KUKA KRL data list: CNC1.dat

&ACCESS RV
DEFDAT CNC1 Public
DECL GLOBAL FRAME gfCNCPoint1[30000]


gfCNCPoint1[1] = {X 300.0000, Y -7.9400, Z 3.0000, A 0.000, B 0.000, C 0.000 }
gfCNCPoint1[2] = {X 300.0000, Y -7.9400, Z 0.0000, A 0.000, B 0.000, C 0.000 }
gfCNCPoint1[3] = {X 300.0000, Y -1.5400, Z 0.0000, A 0.000, B 0.000, C 0.000 }
gfCNCPoint1[4] = {X 0.0000, Y -1.5400, Z 0.0000, A 0.000, B 0.000, C 0.000 }
gfCNCPoint1[5] = {X -1.5400, Y 0.0000, Z 0.0000, A 0.000, B 0.000, C 0.000 }
gfCNCPoint1[6] = {X -1.5400, Y 100.0000, Z 0.0000, A 0.000, B 0.000, C 0.000 }
gfCNCPoint1[7] = {X 0.0000, Y 101.5400, Z 0.0000, A 0.000, B 0.000, C 0.000 }
gfCNCPoint1[8] = {X 600.0000, Y 101.5400, Z 0.0000, A 0.000, B 0.000, C 0.000 }
gfCNCPoint1[9] = {X 601.5400, Y 100.0000, Z 0.0000, A 0.000, B 0.000, C 0.000 }
gfCNCPoint1[10] = {X 601.5400, Y 0.0000, Z 0.0000, A 0.000, B 0.000, C 0.000 }
gfCNCPoint1[11] = {X 600.0000, Y -1.5400, Z 0.0000, A 0.000, B 0.000, C 0.000 }
gfCNCPoint1[12] = {X 300.0000, Y -1.5400, Z 0.0000, A 0.000, B 0.000, C 0.000 }
gfCNCPoint1[13] = {X 300.0000, Y 0.8600, Z 0.0000, A 0.000, B 0.000, C 0.000 }
gfCNCPoint1[14] = {X 0.8600, Y 0.8600, Z 0.0000, A 0.000, B 0.000, C 0.000 }
gfCNCPoint1[15] = {X 0.8600, Y 99.1400, Z 0.0000, A 0.000, B 0.000, C 0.000 }
gfCNCPoint1[16] = {X 599.1400, Y 99.1400, Z 0.0000, A 0.000, B 0.000, C 0.000 }
gfCNCPoint1[17] = {X 599.1400, Y 0.8600, Z 0.0000, A 0.000, B 0.000, C 0.000 }
gfCNCPoint1[18] = {X 300.0000, Y 0.8600, Z 0.0000, A 0.000, B 0.000, C 0.000 }
gfCNCPoint1[19] = {X 300.0000, Y 3.2600, Z 0.0000, A 0.000, B 0.000, C 0.000 }
gfCNCPoint1[20] = {X 3.2600, Y 3.2600, Z 0.0000, A 0.000, B 0.000, C 0.000 }
gfCNCPoint1[21] = {X 3.2600, Y 96.7400, Z 0.0000, A 0.000, B 0.000, C 0.000 }
gfCNCPoint1[22] = {X 596.7400, Y 96.7400, Z 0.0000, A 0.000, B 0.000, C 0.000 }
gfCNCPoint1[23] = {X 596.7400, Y 3.2600, Z 0.0000, A 0.000, B 0.000, C 0.000 }
gfCNCPoint1[24] = {X 300.0000, Y 3.2600, Z 0.0000, A 0.000, B 0.000, C 0.000 }
gfCNCPoint1[25] = {X 300.0000, Y 5.6600, Z 0.0000, A 0.000, B 0.000, C 0.000 }
gfCNCPoint1[26] = {X 5.6600, Y 5.6600, Z 0.0000, A 0.000, B 0.000, C 0.000 }
gfCNCPoint1[27] = {X 5.6600, Y 94.3400, Z 0.0000, A 0.000, B 0.000, C 0.000 }
gfCNCPoint1[28] = {X 594.3400, Y 94.3400, Z 0.0000, A 0.000, B 0.000, C 0.000 }
gfCNCPoint1[29] = {X 594.3400, Y 5.6600, Z 0.0000, A 0.000, B 0.000, C 0.000 }
gfCNCPoint1[30] = {X 300.0000, Y 5.6600, Z 0.0000, A 0.000, B 0.000, C 0.000 }
gfCNCPoint1[31] = {X 300.0000, Y 8.0600, Z 0.0000, A 0.000, B 0.000, C 0.000 }
gfCNCPoint1[32] = {X 8.0600, Y 8.0600, Z 0.0000, A 0.000, B 0.000, C 0.000 }
gfCNCPoint1[33] = {X 8.0600, Y 91.9400, Z 0.0000, A 0.000, B 0.000, C 0.000 }
gfCNCPoint1[34] = {X 591.9400, Y 91.9400, Z 0.0000, A 0.000, B 0.000, C 0.000 }
gfCNCPoint1[35] = {X 591.9400, Y 8.0600, Z 0.0000, A 0.000, B 0.000, C 0.000 }
gfCNCPoint1[36] = {X 300.0000, Y 8.0600, Z 0.0000, A 0.000, B 0.000, C 0.000 }
gfCNCPoint1[37] = {X 300.0000, Y 10.4600, Z 0.0000, A 0.000, B 0.000, C 0.000 }
gfCNCPoint1[38] = {X 10.4600, Y 10.4600, Z 0.0000, A 0.000, B 0.000, C 0.000 }
gfCNCPoint1[39] = {X 10.4600, Y 89.5400, Z 0.0000, A 0.000, B 0.000, C 0.000 }
gfCNCPoint1[40] = {X 589.5400, Y 89.5400, Z 0.0000, A 0.000, B 0.000, C 0.000 }
gfCNCPoint1[41] = {X 589.5400, Y 10.4600, Z 0.0000, A 0.000, B 0.000, C 0.000 }
gfCNCPoint1[42] = {X 300.0000, Y 10.4600, Z 0.0000, A 0.000, B 0.000, C 0.000 }
gfCNCPoint1[43] = {X 300.0000, Y 12.8600, Z 0.0000, A 0.000, B 0.000, C 0.000 }
gfCNCPoint1[44] = {X 12.8600, Y 12.8600, Z 0.0000, A 0.000, B 0.000, C 0.000 }
gfCNCPoint1[45] = {X 12.8600, Y 87.1400, Z 0.0000, A 0.000, B 0.000, C 0.000 }
gfCNCPoint1[46] = {X 587.1400, Y 87.1400, Z 0.0000, A 0.000, B 0.000, C 0.000 }
gfCNCPoint1[47] = {X 587.1400, Y 12.8600, Z 0.0000, A 0.000, B 0.000, C 0.000 }
gfCNCPoint1[48] = {X 300.0000, Y 12.8600, Z 0.0000, A 0.000, B 0.000, C 0.000 }
gfCNCPoint1[49] = {X 300.0000, Y 15.2600, Z 0.0000, A 0.000, B 0.000, C 0.000 }
gfCNCPoint1[50] = {X 15.2600, Y 15.2600, Z 0.0000, A 0.000, B 0.000, C 0.000 }
gfCNCPoint1[51] = {X 15.2600, Y 84.7400, Z 0.0000, A 0.000, B 0.000, C 0.000 }
gfCNCPoint1[52] = {X 584.7400, Y 84.7400, Z 0.0000, A 0.000, B 0.000, C 0.000 }
gfCNCPoint1[53] = {X 584.7400, Y 15.2600, Z 0.0000, A 0.000, B 0.000, C 0.000 }
gfCNCPoint1[54] = {X 300.0000, Y 15.2600, Z 0.0000, A 0.000, B 0.000, C 0.000 }
gfCNCPoint1[55] = {X 300.0000, Y 17.6600, Z 0.0000, A 0.000, B 0.000, C 0.000 }
gfCNCPoint1[56] = {X 17.6600, Y 17.6600, Z 0.0000, A 0.000, B 0.000, C 0.000 }
gfCNCPoint1[57] = {X 17.6600, Y 82.3400, Z 0.0000, A 0.000, B 0.000, C 0.000 }
gfCNCPoint1[58] = {X 582.3400, Y 82.3400, Z 0.0000, A 0.000, B 0.000, C 0.000 }
gfCNCPoint1[59] = {X 582.3400, Y 17.6600, Z 0.0000, A 0.000, B 0.000, C 0.000 }
gfCNCPoint1[60] = {X 300.0000, Y 17.6600, Z 0.0000, A 0.000, B 0.000, C 0.000 }
gfCNCPoint1[61] = {X 300.0000, Y 20.0600, Z 0.0000, A 0.000, B 0.000, C 0.000 }
gfCNCPoint1[62] = {X 20.0600, Y 20.0600, Z 0.0000, A 0.000, B 0.000, C 0.000 }
gfCNCPoint1[63] = {X 20.0600, Y 79.9400, Z 0.0000, A 0.000, B 0.000, C 0.000 }
gfCNCPoint1[64] = {X 579.9400, Y 79.9400, Z 0.0000, A 0.000, B 0.000, C 0.000 }
gfCNCPoint1[65] = {X 579.9400, Y 20.0600, Z 0.0000, A 0.000, B 0.000, C 0.000 }
gfCNCPoint1[66] = {X 300.0000, Y 20.0600, Z 0.0000, A 0.000, B 0.000, C 0.000 }
gfCNCPoint1[67] = {X 300.0000, Y 22.4600, Z 0.0000, A 0.000, B 0.000, C 0.000 }
gfCNCPoint1[68] = {X 22.4600, Y 22.4600, Z 0.0000, A 0.000, B 0.000, C 0.000 }
gfCNCPoint1[69] = {X 22.4600, Y 77.5400, Z 0.0000, A 0.000, B 0.000, C 0.000 }
gfCNCPoint1[70] = {X 577.5400, Y 77.5400, Z 0.0000, A 0.000, B 0.000, C 0.000 }
gfCNCPoint1[71] = {X 577.5400, Y 22.4600, Z 0.0000, A 0.000, B 0.000, C 0.000 }
gfCNCPoint1[72] = {X 300.0000, Y 22.4600, Z 0.0000, A 0.000, B 0.000, C 0.000 }
gfCNCPoint1[73] = {X 300.0000, Y 24.8600, Z 0.0000, A 0.000, B 0.000, C 0.000 }
gfCNCPoint1[74] = {X 24.8600, Y 24.8600, Z 0.0000, A 0.000, B 0.000, C 0.000 }
gfCNCPoint1[75] = {X 24.8600, Y 75.1400, Z 0.0000, A 0.000, B 0.000, C 0.000 }
gfCNCPoint1[76] = {X 575.1400, Y 75.1400, Z 0.0000, A 0.000, B 0.000, C 0.000 }
gfCNCPoint1[77] = {X 575.1400, Y 24.8600, Z 0.0000, A 0.000, B 0.000, C 0.000 }
gfCNCPoint1[78] = {X 300.0000, Y 24.8600, Z 0.0000, A 0.000, B 0.000, C 0.000 }
gfCNCPoint1[79] = {X 300.0000, Y 27.2600, Z 0.0000, A 0.000, B 0.000, C 0.000 }
gfCNCPoint1[80] = {X 27.2600, Y 27.2600, Z 0.0000, A 0.000, B 0.000, C 0.000 }
gfCNCPoint1[81] = {X 27.2600, Y 72.7400, Z 0.0000, A 0.000, B 0.000, C 0.000 }
gfCNCPoint1[82] = {X 572.7400, Y 72.7400, Z 0.0000, A 0.000, B 0.000, C 0.000 }
gfCNCPoint1[83] = {X 572.7400, Y 27.2600, Z 0.0000, A 0.000, B 0.000, C 0.000 }
gfCNCPoint1[84] = {X 300.0000, Y 27.2600, Z 0.0000, A 0.000, B 0.000, C 0.000 }
gfCNCPoint1[85] = {X 300.0000, Y 29.6600, Z 0.0000, A 0.000, B 0.000, C 0.000 }
gfCNCPoint1[86] = {X 29.6600, Y 29.6600, Z 0.0000, A 0.000, B 0.000, C 0.000 }
gfCNCPoint1[87] = {X 29.6600, Y 70.3400, Z 0.0000, A 0.000, B 0.000, C 0.000 }
gfCNCPoint1[88] = {X 570.3400, Y 70.3400, Z 0.0000, A 0.000, B 0.000, C 0.000 }
gfCNCPoint1[89] = {X 570.3400, Y 29.6600, Z 0.0000, A 0.000, B 0.000, C 0.000 }
gfCNCPoint1[90] = {X 300.0000, Y 29.6600, Z 0.0000, A 0.000, B 0.000, C 0.000 }
gfCNCPoint1[91] = {X 300.0000, Y 32.0600, Z 0.0000, A 0.000, B 0.000, C 0.000 }
gfCNCPoint1[92] = {X 32.0600, Y 32.0600, Z 0.0000, A 0.000, B 0.000, C 0.000 }
gfCNCPoint1[93] = {X 32.0600, Y 67.9400, Z 0.0000, A 0.000, B 0.000, C 0.000 }
gfCNCPoint1[94] = {X 567.9400, Y 67.9400, Z 0.0000, A 0.000, B 0.000, C 0.000 }
gfCNCPoint1[95] = {X 567.9400, Y 32.0600, Z 0.0000, A 0.000, B 0.000, C 0.000 }
gfCNCPoint1[96] = {X 300.0000, Y 32.0600, Z 0.0000, A 0.000, B 0.000, C 0.000 }
gfCNCPoint1[97] = {X 300.0000, Y 34.4600, Z 0.0000, A 0.000, B 0.000, C 0.000 }
gfCNCPoint1[98] = {X 34.4600, Y 34.4600, Z 0.0000, A 0.000, B 0.000, C 0.000 }
gfCNCPoint1[99] = {X 34.4600, Y 65.5400, Z 0.0000, A 0.000, B 0.000, C 0.000 }
gfCNCPoint1[100] = {X 565.5400, Y 65.5400, Z 0.0000, A 0.000, B 0.000, C 0.000 }
gfCNCPoint1[101] = {X 565.5400, Y 34.4600, Z 0.0000, A 0.000, B 0.000, C 0.000 }
gfCNCPoint1[102] = {X 300.0000, Y 34.4600, Z 0.0000, A 0.000, B 0.000, C 0.000 }
gfCNCPoint1[103] = {X 300.0000, Y 36.8600, Z 0.0000, A 0.000, B 0.000, C 0.000 }
gfCNCPoint1[104] = {X 36.8600, Y 36.8600, Z 0.0000, A 0.000, B 0.000, C 0.000 }
gfCNCPoint1[105] = {X 36.8600, Y 63.1400, Z 0.0000, A 0.000, B 0.000, C 0.000 }
gfCNCPoint1[106] = {X 563.1400, Y 63.1400, Z 0.0000, A 0.000, B 0.000, C 0.000 }
gfCNCPoint1[107] = {X 563.1400, Y 36.8600, Z 0.0000, A 0.000, B 0.000, C 0.000 }
gfCNCPoint1[108] = {X 300.0000, Y 36.8600, Z 0.0000, A 0.000, B 0.000, C 0.000 }
gfCNCPoint1[109] = {X 300.0000, Y 39.2600, Z 0.0000, A 0.000, B 0.000, C 0.000 }
gfCNCPoint1[110] = {X 39.2600, Y 39.2600, Z 0.0000, A 0.000, B 0.000, C 0.000 }
gfCNCPoint1[111] = {X 39.2600, Y 60.7400, Z 0.0000, A 0.000, B 0.000, C 0.000 }
gfCNCPoint1[112] = {X 560.7400, Y 60.7400, Z 0.0000, A 0.000, B 0.000, C 0.000 }
gfCNCPoint1[113] = {X 560.7400, Y 39.2600, Z 0.0000, A 0.000, B 0.000, C 0.000 }
gfCNCPoint1[114] = {X 300.0000, Y 39.2600, Z 0.0000, A 0.000, B 0.000, C 0.000 }
gfCNCPoint1[115] = {X 300.0000, Y 41.6600, Z 0.0000, A 0.000, B 0.000, C 0.000 }
gfCNCPoint1[116] = {X 41.6600, Y 41.6600, Z 0.0000, A 0.000, B 0.000, C 0.000 }
gfCNCPoint1[117] = {X 41.6600, Y 58.3400, Z 0.0000, A 0.000, B 0.000, C 0.000 }
gfCNCPoint1[118] = {X 558.3400, Y 58.3400, Z 0.0000, A 0.000, B 0.000, C 0.000 }
gfCNCPoint1[119] = {X 558.3400, Y 41.6600, Z 0.0000, A 0.000, B 0.000, C 0.000 }
gfCNCPoint1[120] = {X 300.0000, Y 41.6600, Z 0.0000, A 0.000, B 0.000, C 0.000 }
gfCNCPoint1[121] = {X 300.0000, Y 44.0600, Z 0.0000, A 0.000, B 0.000, C 0.000 }
gfCNCPoint1[122] = {X 44.0600, Y 44.0600, Z 0.0000, A 0.000, B 0.000, C 0.000 }
gfCNCPoint1[123] = {X 44.0600, Y 55.9400, Z 0.0000, A 0.000, B 0.000, C 0.000 }
gfCNCPoint1[124] = {X 555.9400, Y 55.9400, Z 0.0000, A 0.000, B 0.000, C 0.000 }
gfCNCPoint1[125] = {X 555.9400, Y 44.0600, Z 0.0000, A 0.000, B 0.000, C 0.000 }
gfCNCPoint1[126] = {X 300.0000, Y 44.0600, Z 0.0000, A 0.000, B 0.000, C 0.000 }
gfCNCPoint1[127] = {X 300.0000, Y 46.4600, Z 0.0000, A 0.000, B 0.000, C 0.000 }
gfCNCPoint1[128] = {X 46.4600, Y 46.4600, Z 0.0000, A 0.000, B 0.000, C 0.000 }
gfCNCPoint1[129] = {X 46.4600, Y 53.5400, Z 0.0000, A 0.000, B 0.000, C 0.000 }
gfCNCPoint1[130] = {X 553.5400, Y 53.5400, Z 0.0000, A 0.000, B 0.000, C 0.000 }
gfCNCPoint1[131] = {X 553.5400, Y 46.4600, Z 0.0000, A 0.000, B 0.000, C 0.000 }
gfCNCPoint1[132] = {X 300.0000, Y 46.4600, Z 0.0000, A 0.000, B 0.000, C 0.000 }
gfCNCPoint1[133] = {X 300.0000, Y 48.8600, Z 0.0000, A 0.000, B 0.000, C 0.000 }
gfCNCPoint1[134] = {X 48.8600, Y 48.8600, Z 0.0000, A 0.000, B 0.000, C 0.000 }
gfCNCPoint1[135] = {X 48.8600, Y 51.1400, Z 0.0000, A 0.000, B 0.000, C 0.000 }
gfCNCPoint1[136] = {X 551.1400, Y 51.1400, Z 0.0000, A 0.000, B 0.000, C 0.000 }
gfCNCPoint1[137] = {X 551.1400, Y 48.8600, Z 0.0000, A 0.000, B 0.000, C 0.000 }
gfCNCPoint1[138] = {X 300.0000, Y 48.8600, Z 0.0000, A 0.000, B 0.000, C 0.000 }
gfCNCPoint1[139] = {X 300.0000, Y 44.8600, Z 0.0000, A 0.000, B 0.000, C 0.000 }
gfCNCPoint1[140] = {X 300.0000, Y 44.8600, Z 3.0000, A 0.000, B 0.000, C 0.000 }
gfCNCPoint1[141] = {X 300.0000, Y 44.8600, Z 10.0000, A 0.000, B 0.000, C 0.000 }
gfCNCPoint1[142] = {X 607.6965, Y 2.1256, Z 1.6667, A 0.000, B 0.000, C 0.000 }
gfCNCPoint1[143] = {X 607.6965, Y 2.1256, Z -1.3333, A 0.000, B 0.000, C 0.000 }
gfCNCPoint1[144] = {X 603.6965, Y 8.3207, Z -1.3333, A 0.000, B 0.000, C 0.000 }
gfCNCPoint1[145] = {X 603.3199, Y 8.8216, Z -1.3333, A 0.000, B 0.000, C 0.000 }
gfCNCPoint1[146] = {X 602.8760, Y 9.2640, Z -1.3333, A 0.000, B 0.000, C 0.000 }
gfCNCPoint1[147] = {X 602.8760, Y 40.7360, Z -1.3333, A 0.000, B 0.000, C 0.000 }
gfCNCPoint1[148] = {X 603.3199, Y 41.1783, Z -1.3333, A 0.000, B 0.000, C 0.000 }
gfCNCPoint1[149] = {X 603.6965, Y 41.6793, Z -1.3333, A 0.000, B 0.000, C 0.000 }
gfCNCPoint1[150] = {X 607.6965, Y 47.8744, Z -1.3333, A 0.000, B 0.000, C 0.000 }
gfCNCPoint1[151] = {X 607.6965, Y 47.8744, Z 1.6667, A 0.000, B 0.000, C 0.000 }
gfCNCPoint1[152] = {X 607.6965, Y 47.8744, Z 11.0000, A 0.000, B 0.000, C 0.000 }
gfCNCPoint1[153] = {X 607.6965, Y 1.5529, Z 11.0000, A 0.000, B 0.000, C 0.000 }
gfCNCPoint1[154] = {X 607.6965, Y 1.5529, Z 1.6667, A 0.000, B 0.000, C 0.000 }
gfCNCPoint1[155] = {X 607.6965, Y 1.5529, Z -1.3333, A 0.000, B 0.000, C 0.000 }
gfCNCPoint1[156] = {X 603.6965, Y 8.1703, Z -1.3333, A 0.000, B 0.000, C 0.000 }
gfCNCPoint1[157] = {X 603.2890, Y 8.7356, Z -1.3333, A 0.000, B 0.000, C 0.000 }
gfCNCPoint1[158] = {X 602.7960, Y 9.2281, Z -1.3333, A 0.000, B 0.000, C 0.000 }
gfCNCPoint1[159] = {X 602.7960, Y 40.7730, Z -1.3333, A 0.000, B 0.000, C 0.000 }
gfCNCPoint1[160] = {X 603.2890, Y 41.2652, Z -1.3333, A 0.000, B 0.000, C 0.000 }
gfCNCPoint1[161] = {X 603.6965, Y 41.8302, Z -1.3333, A 0.000, B 0.000, C 0.000 }
gfCNCPoint1[162] = {X 607.6965, Y 48.4430, Z -1.3333, A 0.000, B 0.000, C 0.000 }
gfCNCPoint1[163] = {X 607.6965, Y 48.4430, Z 1.6667, A 0.000, B 0.000, C 0.000 }
gfCNCPoint1[164] = {X 607.6965, Y 48.4430, Z 11.0000, A 0.000, B 0.000, C 0.000 }
gfCNCPoint1[165] = {X 607.6965, Y 0.8876, Z 11.0000, A 0.000, B 0.000, C 0.000 }
gfCNCPoint1[166] = {X 607.6965, Y 0.8876, Z 1.6667, A 0.000, B 0.000, C 0.000 }
gfCNCPoint1[167] = {X 607.6965, Y 0.8876, Z -1.3333, A 0.000, B 0.000, C 0.000 }
gfCNCPoint1[168] = {X 603.6965, Y 8.0114, Z -1.3333, A 0.000, B 0.000, C 0.000 }
gfCNCPoint1[169] = {X 603.2600, Y 8.6459, Z -1.3333, A 0.000, B 0.000, C 0.000 }
gfCNCPoint1[170] = {X 602.7160, Y 9.1909, Z -1.3333, A 0.000, B 0.000, C 0.000 }
gfCNCPoint1[171] = {X 602.7160, Y 40.8102, Z -1.3333, A 0.000, B 0.000, C 0.000 }
gfCNCPoint1[172] = {X 603.2600, Y 41.3549, Z -1.3333, A 0.000, B 0.000, C 0.000 }
gfCNCPoint1[173] = {X 603.6965, Y 41.9890, Z -1.3333, A 0.000, B 0.000, C 0.000 }
gfCNCPoint1[174] = {X 607.6965, Y 49.1072, Z -1.3333, A 0.000, B 0.000, C 0.000 }
gfCNCPoint1[175] = {X 607.6965, Y 49.1072, Z 1.6667, A 0.000, B 0.000, C 0.000 }
gfCNCPoint1[176] = {X 607.6965, Y 49.1072, Z 11.0000, A 0.000, B 0.000, C 0.000 }
gfCNCPoint1[177] = {X 607.6950, Y 0.0916, Z 11.0000, A 0.000, B 0.000, C 0.000 }
gfCNCPoint1[178] = {X 607.6950, Y 0.0916, Z 1.6667, A 0.000, B 0.000, C 0.000 }
gfCNCPoint1[179] = {X 607.6950, Y 0.0916, Z -1.3333, A 0.000, B 0.000, C 0.000 }
gfCNCPoint1[180] = {X 603.6965, Y 7.8427, Z -1.3333, A 0.000, B 0.000, C 0.000 }
gfCNCPoint1[181] = {X 603.2333, Y 8.5523, Z -1.3333, A 0.000, B 0.000, C 0.000 }
gfCNCPoint1[182] = {X 602.6360, Y 9.1532, Z -1.3333, A 0.000, B 0.000, C 0.000 }
gfCNCPoint1[183] = {X 602.6360, Y 40.8479, Z -1.3333, A 0.000, B 0.000, C 0.000 }
gfCNCPoint1[184] = {X 603.2333, Y 41.4485, Z -1.3333, A 0.000, B 0.000, C 0.000 }
gfCNCPoint1[185] = {X 603.6965, Y 42.1576, Z -1.3333, A 0.000, B 0.000, C 0.000 }
gfCNCPoint1[186] = {X 607.6965, Y 49.9047, Z -1.3333, A 0.000, B 0.000, C 0.000 }
gfCNCPoint1[187] = {X 607.6965, Y 49.9047, Z 1.6667, A 0.000, B 0.000, C 0.000 }
gfCNCPoint1[188] = {X 607.6965, Y 49.9047, Z 11.0000, A 0.000, B 0.000, C 0.000 }
gfCNCPoint1[189] = {X 607.6538, Y -0.8091, Z 11.0000, A 0.000, B 0.000, C 0.000 }
gfCNCPoint1[190] = {X 607.6538, Y -0.8091, Z 1.6667, A 0.000, B 0.000, C 0.000 }
gfCNCPoint1[191] = {X 607.6538, Y -0.8091, Z -1.3333, A 0.000, B 0.000, C 0.000 }
gfCNCPoint1[192] = {X 603.6965, Y 7.6611, Z -1.3333, A 0.000, B 0.000, C 0.000 }
gfCNCPoint1[193] = {X 603.2067, Y 8.4567, Z -1.3333, A 0.000, B 0.000, C 0.000 }
gfCNCPoint1[194] = {X 602.5488, Y 9.1200, Z -1.3333, A 0.000, B 0.000, C 0.000 }
gfCNCPoint1[195] = {X 602.5560, Y 9.1532, Z -1.3333, A 0.000, B 0.000, C 0.000 }
gfCNCPoint1[196] = {X 602.5560, Y 40.8856, Z -1.3333, A 0.000, B 0.000, C 0.000 }
gfCNCPoint1[197] = {X 602.6236, Y 40.9413, Z -1.3333, A 0.000, B 0.000, C 0.000 }
gfCNCPoint1[198] = {X 603.2364, Y 41.5815, Z -1.3333, A 0.000, B 0.000, C 0.000 }
gfCNCPoint1[199] = {X 603.6965, Y 42.3389, Z -1.3333, A 0.000, B 0.000, C 0.000 }
gfCNCPoint1[200] = {X 607.6965, Y 50.9003, Z -1.3333, A 0.000, B 0.000, C 0.000 }
gfCNCPoint1[201] = {X 607.6965, Y 50.9003, Z 1.6667, A 0.000, B 0.000, C 0.000 }
gfCNCPoint1[202] = {X 607.6965, Y 50.9003, Z 11.0000, A 0.000, B 0.000, C 0.000 }
gfCNCPoint1[203] = {X 607.4989, Y -1.7333, Z 11.0000, A 0.000, B 0.000, C 0.000 }
gfCNCPoint1[204] = {X 607.4989, Y -1.7333, Z 1.6667, A 0.000, B 0.000, C 0.000 }
gfCNCPoint1[205] = {X 607.4989, Y -1.7333, Z -1.3333, A 0.000, B 0.000, C 0.000 }
gfCNCPoint1[206] = {X 603.6965, Y 7.4625, Z -1.3333, A 0.000, B 0.000, C 0.000 }
gfCNCPoint1[207] = {X 603.3768, Y 8.0782, Z -1.3333, A 0.000, B 0.000, C 0.000 }
gfCNCPoint1[208] = {X 602.9556, Y 8.6294, Z -1.3333, A 0.000, B 0.000, C 0.000 }
gfCNCPoint1[209] = {X 602.4454, Y 9.0995, Z -1.3333, A 0.000, B 0.000, C 0.000 }
gfCNCPoint1[210] = {X 602.4760, Y 9.1532, Z -1.3333, A 0.000, B 0.000, C 0.000 }
gfCNCPoint1[211] = {X 602.4760, Y 40.9232, Z -1.3333, A 0.000, B 0.000, C 0.000 }
gfCNCPoint1[212] = {X 602.5724, Y 41.0028, Z -1.3333, A 0.000, B 0.000, C 0.000 }
gfCNCPoint1[213] = {X 603.2270, Y 41.7024, Z -1.3333, A 0.000, B 0.000, C 0.000 }
gfCNCPoint1[214] = {X 603.6965, Y 42.5375, Z -1.3333, A 0.000, B 0.000, C 0.000 }
gfCNCPoint1[215] = {X 607.6965, Y 52.2111, Z -1.3333, A 0.000, B 0.000, C 0.000 }
gfCNCPoint1[216] = {X 607.6965, Y 52.2111, Z 1.6667, A 0.000, B 0.000, C 0.000 }
gfCNCPoint1[217] = {X 607.6965, Y 52.2111, Z 11.0000, A 0.000, B 0.000, C 0.000 }
gfCNCPoint1[218] = {X 492.1926, Y 19.7807, Z 11.0000, A 0.000, B 0.000, C 0.000 }
gfCNCPoint1[219] = {X 492.1926, Y 19.7807, Z 2.5000, A 0.000, B 0.000, C 0.000 }
gfCNCPoint1[220] = {X 487.6645, Y 19.7797, Z 1.2867, A 0.000, B 0.000, C 0.000 }
gfCNCPoint1[221] = {X 486.9699, Y 19.7845, Z 1.1006, A 0.000, B 0.000, C 0.000 }
gfCNCPoint1[222] = {X 486.2675, Y 19.7831, Z 0.9124, A 0.000, B 0.000, C 0.000 }
gfCNCPoint1[223] = {X 485.4752, Y 19.8882, Z 0.6982, A 0.000, B 0.000, C 0.000 }
gfCNCPoint1[224] = {X 484.7975, Y 20.0727, Z 0.5100, A 0.000, B 0.000, C 0.000 }
gfCNCPoint1[225] = {X 484.6636, Y 20.1091, Z 0.4728, A 0.000, B 0.000, C 0.000 }
gfCNCPoint1[226] = {X 484.6335, Y 20.1374, Z 0.4618, A 0.000, B 0.000, C 0.000 }
gfCNCPoint1[227] = {X 484.5885, Y 20.2686, Z 0.4246, A 0.000, B 0.000, C 0.000 }
gfCNCPoint1[228] = {X 484.4391, Y 20.7049, Z 0.3010, A 0.000, B 0.000, C 0.000 }
gfCNCPoint1[229] = {X 484.4030, Y 21.9111, Z -0.0223, A 0.000, B 0.000, C 0.000 }
gfCNCPoint1[230] = {X 484.5262, Y 22.3556, Z -0.1459, A 0.000, B 0.000, C 0.000 }
gfCNCPoint1[231] = {X 484.6980, Y 22.4116, Z -0.1943, A 0.000, B 0.000, C 0.000 }
gfCNCPoint1[232] = {X 484.8776, Y 22.4314, Z -0.2427, A 0.000, B 0.000, C 0.000 }
gfCNCPoint1[233] = {X 486.0306, Y 22.5560, Z -0.5535, A 0.000, B 0.000, C 0.000 }
gfCNCPoint1[234] = {X 487.1449, Y 22.5560, Z -0.8521, A 0.000, B 0.000, C 0.000 }
gfCNCPoint1[235] = {X 488.9410, Y 22.5560, Z -1.3333, A 0.000, B 0.000, C 0.000 }
gfCNCPoint1[236] = {X 493.3690, Y 22.5560, Z -1.3333, A 0.000, B 0.000, C 0.000 }
gfCNCPoint1[237] = {X 493.3690, Y 19.7809, Z -1.3333, A 0.000, B 0.000, C 0.000 }
gfCNCPoint1[238] = {X 487.6645, Y 19.7797, Z -1.3333, A 0.000, B 0.000, C 0.000 }
gfCNCPoint1[239] = {X 486.9699, Y 19.7845, Z -1.3333, A 0.000, B 0.000, C 0.000 }
gfCNCPoint1[240] = {X 485.8740, Y 19.8557, Z -1.3333, A 0.000, B 0.000, C 0.000 }
gfCNCPoint1[241] = {X 484.7975, Y 20.0727, Z -1.3333, A 0.000, B 0.000, C 0.000 }
gfCNCPoint1[242] = {X 484.6687, Y 20.1447, Z -1.3333, A 0.000, B 0.000, C 0.000 }
gfCNCPoint1[243] = {X 484.5885, Y 20.2686, Z -1.3333, A 0.000, B 0.000, C 0.000 }
gfCNCPoint1[244] = {X 484.4277, Y 20.9554, Z -1.3333, A 0.000, B 0.000, C 0.000 }
gfCNCPoint1[245] = {X 484.4067, Y 21.6604, Z -1.3333, A 0.000, B 0.000, C 0.000 }
gfCNCPoint1[246] = {X 484.5262, Y 22.3556, Z -1.3333, A 0.000, B 0.000, C 0.000 }
gfCNCPoint1[247] = {X 484.7000, Y 22.4025, Z -1.3333, A 0.000, B 0.000, C 0.000 }
gfCNCPoint1[248] = {X 484.8776, Y 22.4314, Z -1.3333, A 0.000, B 0.000, C 0.000 }
gfCNCPoint1[249] = {X 486.0096, Y 22.5249, Z -1.3333, A 0.000, B 0.000, C 0.000 }
gfCNCPoint1[250] = {X 487.1449, Y 22.5560, Z -1.3333, A 0.000, B 0.000, C 0.000 }
gfCNCPoint1[251] = {X 488.9410, Y 22.5560, Z -1.3333, A 0.000, B 0.000, C 0.000 }
gfCNCPoint1[252] = {X 484.9562, Y 22.2874, Z -1.3333, A 0.000, B 0.000, C 0.000 }
gfCNCPoint1[253] = {X 488.9410, Y 22.6360, Z -1.3333, A 0.000, B 0.000, C 0.000 }
gfCNCPoint1[254] = {X 493.4490, Y 22.6360, Z -1.3333, A 0.000, B 0.000, C 0.000 }
gfCNCPoint1[255] = {X 493.4490, Y 19.7009, Z -1.3333, A 0.000, B 0.000, C 0.000 }
gfCNCPoint1[256] = {X 487.6642, Y 19.6997, Z -1.3333, A 0.000, B 0.000, C 0.000 }
gfCNCPoint1[257] = {X 486.9714, Y 19.7045, Z -1.3333, A 0.000, B 0.000, C 0.000 }
gfCNCPoint1[258] = {X 485.8642, Y 19.7763, Z -1.3333, A 0.000, B 0.000, C 0.000 }
gfCNCPoint1[259] = {X 484.7765, Y 19.9955, Z -1.3333, A 0.000, B 0.000, C 0.000 }
gfCNCPoint1[260] = {X 484.6139, Y 20.0863, Z -1.3333, A 0.000, B 0.000, C 0.000 }
gfCNCPoint1[261] = {X 484.5129, Y 20.2427, Z -1.3333, A 0.000, B 0.000, C 0.000 }
gfCNCPoint1[262] = {X 484.3466, Y 20.9591, Z -1.3333, A 0.000, B 0.000, C 0.000 }
gfCNCPoint1[263] = {X 484.3290, Y 21.6943, Z -1.3333, A 0.000, B 0.000, C 0.000 }
gfCNCPoint1[264] = {X 484.4607, Y 22.4179, Z -1.3333, A 0.000, B 0.000, C 0.000 }
gfCNCPoint1[265] = {X 484.6621, Y 22.4761, Z -1.3333, A 0.000, B 0.000, C 0.000 }
gfCNCPoint1[266] = {X 484.8689, Y 22.5109, Z -1.3333, A 0.000, B 0.000, C 0.000 }
gfCNCPoint1[267] = {X 486.0052, Y 22.6047, Z -1.3333, A 0.000, B 0.000, C 0.000 }
gfCNCPoint1[268] = {X 487.1449, Y 22.6360, Z -1.3333, A 0.000, B 0.000, C 0.000 }
gfCNCPoint1[269] = {X 488.9410, Y 22.6360, Z -1.3333, A 0.000, B 0.000, C 0.000 }
gfCNCPoint1[270] = {X 492.9257, Y 22.2874, Z -1.3333, A 0.000, B 0.000, C 0.000 }
gfCNCPoint1[271] = {X 484.9562, Y 22.3674, Z -1.3333, A 0.000, B 0.000, C 0.000 }
gfCNCPoint1[272] = {X 488.9410, Y 22.7160, Z -1.3333, A 0.000, B 0.000, C 0.000 }
gfCNCPoint1[273] = {X 493.5290, Y 22.7160, Z -1.3333, A 0.000, B 0.000, C 0.000 }
gfCNCPoint1[274] = {X 493.5290, Y 19.6209, Z -1.3333, A 0.000, B 0.000, C 0.000 }
gfCNCPoint1[275] = {X 487.6640, Y 19.6197, Z -1.3333, A 0.000, B 0.000, C 0.000 }
gfCNCPoint1[276] = {X 486.9712, Y 19.6245, Z -1.3333, A 0.000, B 0.000, C 0.000 }
gfCNCPoint1[277] = {X 485.8535, Y 19.6971, Z -1.3333, A 0.000, B 0.000, C 0.000 }
gfCNCPoint1[278] = {X 484.7555, Y 19.9183, Z -1.3333, A 0.000, B 0.000, C 0.000 }
gfCNCPoint1[279] = {X 484.5592, Y 20.0279, Z -1.3333, A 0.000, B 0.000, C 0.000 }
gfCNCPoint1[280] = {X 484.4372, Y 20.2167, Z -1.3333, A 0.000, B 0.000, C 0.000 }
gfCNCPoint1[281] = {X 484.2655, Y 20.9625, Z -1.3333, A 0.000, B 0.000, C 0.000 }
gfCNCPoint1[282] = {X 484.2514, Y 21.7276, Z -1.3333, A 0.000, B 0.000, C 0.000 }
gfCNCPoint1[283] = {X 484.3954, Y 22.4792, Z -1.3333, A 0.000, B 0.000, C 0.000 }
gfCNCPoint1[284] = {X 484.6243, Y 22.5494, Z -1.3333, A 0.000, B 0.000, C 0.000 }
gfCNCPoint1[285] = {X 484.8601, Y 22.5904, Z -1.3333, A 0.000, B 0.000, C 0.000 }
gfCNCPoint1[286] = {X 486.0008, Y 22.6846, Z -1.3333, A 0.000, B 0.000, C 0.000 }
gfCNCPoint1[287] = {X 487.1449, Y 22.7160, Z -1.3333, A 0.000, B 0.000, C 0.000 }
gfCNCPoint1[288] = {X 488.9410, Y 22.7160, Z -1.3333, A 0.000, B 0.000, C 0.000 }
gfCNCPoint1[289] = {X 492.9257, Y 22.3674, Z -1.3333, A 0.000, B 0.000, C 0.000 }
gfCNCPoint1[290] = {X 484.9562, Y 22.4474, Z -1.3333, A 0.000, B 0.000, C 0.000 }
gfCNCPoint1[291] = {X 488.9410, Y 22.7960, Z -1.3333, A 0.000, B 0.000, C 0.000 }
gfCNCPoint1[292] = {X 493.6090, Y 22.7960, Z -1.3333, A 0.000, B 0.000, C 0.000 }
gfCNCPoint1[293] = {X 493.6090, Y 19.5409, Z -1.3333, A 0.000, B 0.000, C 0.000 }
gfCNCPoint1[294] = {X 487.6637, Y 19.5397, Z -1.3333, A 0.000, B 0.000, C 0.000 }
gfCNCPoint1[295] = {X 486.9711, Y 19.5445, Z -1.3333, A 0.000, B 0.000, C 0.000 }
gfCNCPoint1[296] = {X 485.8428, Y 19.6178, Z -1.3333, A 0.000, B 0.000, C 0.000 }
gfCNCPoint1[297] = {X 484.7345, Y 19.8411, Z -1.3333, A 0.000, B 0.000, C 0.000 }
gfCNCPoint1[298] = {X 484.5045, Y 19.9696, Z -1.3333, A 0.000, B 0.000, C 0.000 }
gfCNCPoint1[299] = {X 484.3615, Y 20.1908, Z -1.3333, A 0.000, B 0.000, C 0.000 }
gfCNCPoint1[300] = {X 484.1846, Y 20.9657, Z -1.3333, A 0.000, B 0.000, C 0.000 }
gfCNCPoint1[301] = {X 484.1740, Y 21.7605, Z -1.3333, A 0.000, B 0.000, C 0.000 }
gfCNCPoint1[302] = {X 484.3303, Y 22.5398, Z -1.3333, A 0.000, B 0.000, C 0.000 }
gfCNCPoint1[303] = {X 484.5864, Y 22.6225, Z -1.3333, A 0.000, B 0.000, C 0.000 }
gfCNCPoint1[304] = {X 484.8513, Y 22.6699, Z -1.3333, A 0.000, B 0.000, C 0.000 }
gfCNCPoint1[305] = {X 485.9964, Y 22.7645, Z -1.3333, A 0.000, B 0.000, C 0.000 }
gfCNCPoint1[306] = {X 487.1449, Y 22.7960, Z -1.3333, A 0.000, B 0.000, C 0.000 }
gfCNCPoint1[307] = {X 488.9410, Y 22.7960, Z -1.3333, A 0.000, B 0.000, C 0.000 }
gfCNCPoint1[308] = {X 492.9257, Y 22.4474, Z -1.3333, A 0.000, B 0.000, C 0.000 }
gfCNCPoint1[309] = {X 484.9562, Y 22.5274, Z -1.3333, A 0.000, B 0.000, C 0.000 }
gfCNCPoint1[310] = {X 488.9410, Y 22.8760, Z -1.3333, A 0.000, B 0.000, C 0.000 }
gfCNCPoint1[311] = {X 493.6890, Y 22.8760, Z -1.3333, A 0.000, B 0.000, C 0.000 }
gfCNCPoint1[312] = {X 493.6890, Y 19.4610, Z -1.3333, A 0.000, B 0.000, C 0.000 }
gfCNCPoint1[313] = {X 487.6634, Y 19.4597, Z -1.3333, A 0.000, B 0.000, C 0.000 }
gfCNCPoint1[314] = {X 486.9709, Y 19.4645, Z -1.3333, A 0.000, B 0.000, C 0.000 }
gfCNCPoint1[315] = {X 485.8321, Y 19.5385, Z -1.3333, A 0.000, B 0.000, C 0.000 }
gfCNCPoint1[316] = {X 484.7134, Y 19.7639, Z -1.3333, A 0.000, B 0.000, C 0.000 }
gfCNCPoint1[317] = {X 484.4498, Y 19.9112, Z -1.3333, A 0.000, B 0.000, C 0.000 }
gfCNCPoint1[318] = {X 484.2858, Y 20.1649, Z -1.3333, A 0.000, B 0.000, C 0.000 }
gfCNCPoint1[319] = {X 484.1037, Y 20.9687, Z -1.3333, A 0.000, B 0.000, C 0.000 }
gfCNCPoint1[320] = {X 484.0968, Y 21.7929, Z -1.3333, A 0.000, B 0.000, C 0.000 }
gfCNCPoint1[321] = {X 484.2655, Y 22.5997, Z -1.3333, A 0.000, B 0.000, C 0.000 }
gfCNCPoint1[322] = {X 484.5486, Y 22.6954, Z -1.3333, A 0.000, B 0.000, C 0.000 }
gfCNCPoint1[323] = {X 484.8425, Y 22.7495, Z -1.3333, A 0.000, B 0.000, C 0.000 }
gfCNCPoint1[324] = {X 485.9920, Y 22.8444, Z -1.3333, A 0.000, B 0.000, C 0.000 }
gfCNCPoint1[325] = {X 487.1449, Y 22.8760, Z -1.3333, A 0.000, B 0.000, C 0.000 }
gfCNCPoint1[326] = {X 488.9410, Y 22.8760, Z -1.3333, A 0.000, B 0.000, C 0.000 }
gfCNCPoint1[327] = {X 492.9257, Y 22.5274, Z -1.3333, A 0.000, B 0.000, C 0.000 }
gfCNCPoint1[328] = {X 484.9562, Y 22.6074, Z -1.3333, A 0.000, B 0.000, C 0.000 }
gfCNCPoint1[329] = {X 488.9410, Y 22.9560, Z -1.3333, A 0.000, B 0.000, C 0.000 }
gfCNCPoint1[330] = {X 493.7690, Y 22.9560, Z -1.3333, A 0.000, B 0.000, C 0.000 }
gfCNCPoint1[331] = {X 493.7704, Y 19.3810, Z -1.3333, A 0.000, B 0.000, C 0.000 }
gfCNCPoint1[332] = {X 487.6632, Y 19.3797, Z -1.3333, A 0.000, B 0.000, C 0.000 }
gfCNCPoint1[333] = {X 486.9707, Y 19.3845, Z -1.3333, A 0.000, B 0.000, C 0.000 }
gfCNCPoint1[334] = {X 485.8214, Y 19.4592, Z -1.3333, A 0.000, B 0.000, C 0.000 }
gfCNCPoint1[335] = {X 484.6924, Y 19.6867, Z -1.3333, A 0.000, B 0.000, C 0.000 }
gfCNCPoint1[336] = {X 484.3950, Y 19.8529, Z -1.3333, A 0.000, B 0.000, C 0.000 }
gfCNCPoint1[337] = {X 484.2101, Y 20.1390, Z -1.3333, A 0.000, B 0.000, C 0.000 }
gfCNCPoint1[338] = {X 484.0228, Y 20.9716, Z -1.3333, A 0.000, B 0.000, C 0.000 }
gfCNCPoint1[339] = {X 484.0196, Y 21.8249, Z -1.3333, A 0.000, B 0.000, C 0.000 }
gfCNCPoint1[340] = {X 484.2007, Y 22.6589, Z -1.3333, A 0.000, B 0.000, C 0.000 }
gfCNCPoint1[341] = {X 484.5108, Y 22.7681, Z -1.3333, A 0.000, B 0.000, C 0.000 }
gfCNCPoint1[342] = {X 484.8338, Y 22.8290, Z -1.3333, A 0.000, B 0.000, C 0.000 }
gfCNCPoint1[343] = {X 485.9876, Y 22.9243, Z -1.3333, A 0.000, B 0.000, C 0.000 }
gfCNCPoint1[344] = {X 487.1449, Y 22.9560, Z -1.3333, A 0.000, B 0.000, C 0.000 }
gfCNCPoint1[345] = {X 488.9410, Y 22.9560, Z -1.3333, A 0.000, B 0.000, C 0.000 }
gfCNCPoint1[346] = {X 492.9410, Y 22.9560, Z -1.3333, A 0.000, B 0.000, C 0.000 }
gfCNCPoint1[347] = {X 492.9410, Y 22.9560, Z 1.6667, A 0.000, B 0.000, C 0.000 }
gfCNCPoint1[348] = {X 492.9410, Y 22.9560, Z 11.0000, A 0.000, B 0.000, C 0.000 }
gfCNCPoint1[349] = {X 448.7112, Y 19.7808, Z 11.0000, A 0.000, B 0.000, C 0.000 }
gfCNCPoint1[350] = {X 448.7112, Y 19.7808, Z 2.5000, A 0.000, B 0.000, C 0.000 }
gfCNCPoint1[351] = {X 444.0413, Y 19.7804, Z 1.2487, A 0.000, B 0.000, C 0.000 }
gfCNCPoint1[352] = {X 443.3490, Y 19.7966, Z 1.0631, A 0.000, B 0.000, C 0.000 }
gfCNCPoint1[353] = {X 442.7479, Y 19.8038, Z 0.9021, A 0.000, B 0.000, C 0.000 }
gfCNCPoint1[354] = {X 442.0372, Y 19.9269, Z 0.7088, A 0.000, B 0.000, C 0.000 }
gfCNCPoint1[355] = {X 441.4687, Y 20.1223, Z 0.5477, A 0.000, B 0.000, C 0.000 }
gfCNCPoint1[356] = {X 441.3656, Y 20.1577, Z 0.5185, A 0.000, B 0.000, C 0.000 }
gfCNCPoint1[357] = {X 441.3325, Y 20.2616, Z 0.4893, A 0.000, B 0.000, C 0.000 }
gfCNCPoint1[358] = {X 441.1876, Y 20.7170, Z 0.3612, A 0.000, B 0.000, C 0.000 }
gfCNCPoint1[359] = {X 441.1538, Y 21.8894, Z 0.0470, A 0.000, B 0.000, C 0.000 }
gfCNCPoint1[360] = {X 441.2723, Y 22.3524, Z -0.0811, A 0.000, B 0.000, C 0.000 }
gfCNCPoint1[361] = {X 441.5005, Y 22.4271, Z -0.1454, A 0.000, B 0.000, C 0.000 }
gfCNCPoint1[362] = {X 442.9760, Y 22.5632, Z -0.5425, A 0.000, B 0.000, C 0.000 }
gfCNCPoint1[363] = {X 443.1481, Y 22.5702, Z -0.5886, A 0.000, B 0.000, C 0.000 }
gfCNCPoint1[364] = {X 444.3942, Y 22.5560, Z -0.9225, A 0.000, B 0.000, C 0.000 }
gfCNCPoint1[365] = {X 445.9273, Y 22.5560, Z -1.3333, A 0.000, B 0.000, C 0.000 }
gfCNCPoint1[366] = {X 450.1184, Y 22.5560, Z -1.3333, A 0.000, B 0.000, C 0.000 }
gfCNCPoint1[367] = {X 450.1184, Y 19.7809, Z -1.3333, A 0.000, B 0.000, C 0.000 }
gfCNCPoint1[368] = {X 444.0413, Y 19.7804, Z -1.3333, A 0.000, B 0.000, C 0.000 }
gfCNCPoint1[369] = {X 443.3490, Y 19.7966, Z -1.3333, A 0.000, B 0.000, C 0.000 }
gfCNCPoint1[370] = {X 442.3958, Y 19.8843, Z -1.3333, A 0.000, B 0.000, C 0.000 }
gfCNCPoint1[371] = {X 441.4687, Y 20.1223, Z -1.3333, A 0.000, B 0.000, C 0.000 }
gfCNCPoint1[372] = {X 441.3841, Y 20.1758, Z -1.3333, A 0.000, B 0.000, C 0.000 }
gfCNCPoint1[373] = {X 441.3325, Y 20.2616, Z -1.3333, A 0.000, B 0.000, C 0.000 }
gfCNCPoint1[374] = {X 441.1820, Y 20.9507, Z -1.3333, A 0.000, B 0.000, C 0.000 }
gfCNCPoint1[375] = {X 441.1617, Y 21.6558, Z -1.3333, A 0.000, B 0.000, C 0.000 }
gfCNCPoint1[376] = {X 441.2723, Y 22.3524, Z -1.3333, A 0.000, B 0.000, C 0.000 }
gfCNCPoint1[377] = {X 441.5032, Y 22.4139, Z -1.3333, A 0.000, B 0.000, C 0.000 }
gfCNCPoint1[378] = {X 441.7395, Y 22.4492, Z -1.3333, A 0.000, B 0.000, C 0.000 }
gfCNCPoint1[379] = {X 443.0655, Y 22.5370, Z -1.3333, A 0.000, B 0.000, C 0.000 }
gfCNCPoint1[380] = {X 444.3942, Y 22.5560, Z -1.3333, A 0.000, B 0.000, C 0.000 }
gfCNCPoint1[381] = {X 445.9273, Y 22.5560, Z -1.3333, A 0.000, B 0.000, C 0.000 }
gfCNCPoint1[382] = {X 441.9425, Y 22.2874, Z -1.3333, A 0.000, B 0.000, C 0.000 }
gfCNCPoint1[383] = {X 445.9273, Y 22.6360, Z -1.3333, A 0.000, B 0.000, C 0.000 }
gfCNCPoint1[384] = {X 450.1984, Y 22.6360, Z -1.3333, A 0.000, B 0.000, C 0.000 }
gfCNCPoint1[385] = {X 450.1984, Y 19.7009, Z -1.3333, A 0.000, B 0.000, C 0.000 }
gfCNCPoint1[386] = {X 444.0404, Y 19.7004, Z -1.3333, A 0.000, B 0.000, C 0.000 }
gfCNCPoint1[387] = {X 443.3498, Y 19.7166, Z -1.3333, A 0.000, B 0.000, C 0.000 }
gfCNCPoint1[388] = {X 442.3831, Y 19.8053, Z -1.3333, A 0.000, B 0.000, C 0.000 }
gfCNCPoint1[389] = {X 441.4427, Y 20.0466, Z -1.3333, A 0.000, B 0.000, C 0.000 }
gfCNCPoint1[390] = {X 441.3269, Y 20.1198, Z -1.3333, A 0.000, B 0.000, C 0.000 }
gfCNCPoint1[391] = {X 441.2563, Y 20.2373, Z -1.3333, A 0.000, B 0.000, C 0.000 }
gfCNCPoint1[392] = {X 441.1009, Y 20.9554, Z -1.3333, A 0.000, B 0.000, C 0.000 }
gfCNCPoint1[393] = {X 441.0838, Y 21.6899, Z -1.3333, A 0.000, B 0.000, C 0.000 }
gfCNCPoint1[394] = {X 441.2058, Y 22.4144, Z -1.3333, A 0.000, B 0.000, C 0.000 }
gfCNCPoint1[395] = {X 441.4655, Y 22.4877, Z -1.3333, A 0.000, B 0.000, C 0.000 }
gfCNCPoint1[396] = {X 441.7322, Y 22.5288, Z -1.3333, A 0.000, B 0.000, C 0.000 }
gfCNCPoint1[397] = {X 443.0609, Y 22.6168, Z -1.3333, A 0.000, B 0.000, C 0.000 }
gfCNCPoint1[398] = {X 444.3924, Y 22.6360, Z -1.3333, A 0.000, B 0.000, C 0.000 }
gfCNCPoint1[399] = {X 445.9273, Y 22.6360, Z -1.3333, A 0.000, B 0.000, C 0.000 }
gfCNCPoint1[400] = {X 449.9121, Y 22.2874, Z -1.3333, A 0.000, B 0.000, C 0.000 }
gfCNCPoint1[401] = {X 441.9425, Y 22.3674, Z -1.3333, A 0.000, B 0.000, C 0.000 }
gfCNCPoint1[402] = {X 445.9273, Y 22.7160, Z -1.3333, A 0.000, B 0.000, C 0.000 }
gfCNCPoint1[403] = {X 450.2784, Y 22.7160, Z -1.3333, A 0.000, B 0.000, C 0.000 }
gfCNCPoint1[404] = {X 450.2784, Y 19.6210, Z -1.3333, A 0.000, B 0.000, C 0.000 }
gfCNCPoint1[405] = {X 444.0395, Y 19.6204, Z -1.3333, A 0.000, B 0.000, C 0.000 }
gfCNCPoint1[406] = {X 443.3484, Y 19.6366, Z -1.3333, A 0.000, B 0.000, C 0.000 }
gfCNCPoint1[407] = {X 442.3692, Y 19.7265, Z -1.3333, A 0.000, B 0.000, C 0.000 }
gfCNCPoint1[408] = {X 441.4167, Y 19.9709, Z -1.3333, A 0.000, B 0.000, C 0.000 }
gfCNCPoint1[409] = {X 441.2697, Y 20.0639, Z -1.3333, A 0.000, B 0.000, C 0.000 }
gfCNCPoint1[410] = {X 441.1801, Y 20.2130, Z -1.3333, A 0.000, B 0.000, C 0.000 }
gfCNCPoint1[411] = {X 441.0198, Y 20.9598, Z -1.3333, A 0.000, B 0.000, C 0.000 }
gfCNCPoint1[412] = {X 441.0062, Y 21.7235, Z -1.3333, A 0.000, B 0.000, C 0.000 }
gfCNCPoint1[413] = {X 441.1397, Y 22.4756, Z -1.3333, A 0.000, B 0.000, C 0.000 }
gfCNCPoint1[414] = {X 441.4279, Y 22.5613, Z -1.3333, A 0.000, B 0.000, C 0.000 }
gfCNCPoint1[415] = {X 441.7248, Y 22.6085, Z -1.3333, A 0.000, B 0.000, C 0.000 }
gfCNCPoint1[416] = {X 443.0575, Y 22.6967, Z -1.3333, A 0.000, B 0.000, C 0.000 }
gfCNCPoint1[417] = {X 444.3929, Y 22.7160, Z -1.3333, A 0.000, B 0.000, C 0.000 }
gfCNCPoint1[418] = {X 445.9273, Y 22.7160, Z -1.3333, A 0.000, B 0.000, C 0.000 }
gfCNCPoint1[419] = {X 449.9121, Y 22.3674, Z -1.3333, A 0.000, B 0.000, C 0.000 }
gfCNCPoint1[420] = {X 441.9425, Y 22.4474, Z -1.3333, A 0.000, B 0.000, C 0.000 }
gfCNCPoint1[421] = {X 445.9273, Y 22.7960, Z -1.3333, A 0.000, B 0.000, C 0.000 }
gfCNCPoint1[422] = {X 450.3584, Y 22.7960, Z -1.3333, A 0.000, B 0.000, C 0.000 }
gfCNCPoint1[423] = {X 450.3584, Y 19.5410, Z -1.3333, A 0.000, B 0.000, C 0.000 }
gfCNCPoint1[424] = {X 444.0385, Y 19.5404, Z -1.3333, A 0.000, B 0.000, C 0.000 }
gfCNCPoint1[425] = {X 443.3470, Y 19.5566, Z -1.3333, A 0.000, B 0.000, C 0.000 }
gfCNCPoint1[426] = {X 442.3553, Y 19.6478, Z -1.3333, A 0.000, B 0.000, C 0.000 }
gfCNCPoint1[427] = {X 441.3907, Y 19.8953, Z -1.3333, A 0.000, B 0.000, C 0.000 }
gfCNCPoint1[428] = {X 441.2125, Y 20.0080, Z -1.3333, A 0.000, B 0.000, C 0.000 }
gfCNCPoint1[429] = {X 441.1038, Y 20.1888, Z -1.3333, A 0.000, B 0.000, C 0.000 }
gfCNCPoint1[430] = {X 440.9388, Y 20.9641, Z -1.3333, A 0.000, B 0.000, C 0.000 }
gfCNCPoint1[431] = {X 440.9286, Y 21.7568, Z -1.3333, A 0.000, B 0.000, C 0.000 }
gfCNCPoint1[432] = {X 441.0737, Y 22.5361, Z -1.3333, A 0.000, B 0.000, C 0.000 }
gfCNCPoint1[433] = {X 441.3903, Y 22.6347, Z -1.3333, A 0.000, B 0.000, C 0.000 }
gfCNCPoint1[434] = {X 441.7175, Y 22.6881, Z -1.3333, A 0.000, B 0.000, C 0.000 }
gfCNCPoint1[435] = {X 443.0540, Y 22.7767, Z -1.3333, A 0.000, B 0.000, C 0.000 }
gfCNCPoint1[436] = {X 444.3933, Y 22.7960, Z -1.3333, A 0.000, B 0.000, C 0.000 }
gfCNCPoint1[437] = {X 445.9273, Y 22.7960, Z -1.3333, A 0.000, B 0.000, C 0.000 }
gfCNCPoint1[438] = {X 449.9121, Y 22.4474, Z -1.3333, A 0.000, B 0.000, C 0.000 }
gfCNCPoint1[439] = {X 441.9425, Y 22.5274, Z -1.3333, A 0.000, B 0.000, C 0.000 }
gfCNCPoint1[440] = {X 445.9273, Y 22.8760, Z -1.3333, A 0.000, B 0.000, C 0.000 }
gfCNCPoint1[441] = {X 450.4384, Y 22.8760, Z -1.3333, A 0.000, B 0.000, C 0.000 }
gfCNCPoint1[442] = {X 450.4384, Y 19.4610, Z -1.3333, A 0.000, B 0.000, C 0.000 }
gfCNCPoint1[443] = {X 444.0376, Y 19.4604, Z -1.3333, A 0.000, B 0.000, C 0.000 }
gfCNCPoint1[444] = {X 443.3456, Y 19.4766, Z -1.3333, A 0.000, B 0.000, C 0.000 }
gfCNCPoint1[445] = {X 442.3415, Y 19.5690, Z -1.3333, A 0.000, B 0.000, C 0.000 }
gfCNCPoint1[446] = {X 441.3647, Y 19.8196, Z -1.3333, A 0.000, B 0.000, C 0.000 }
gfCNCPoint1[447] = {X 441.1553, Y 19.9521, Z -1.3333, A 0.000, B 0.000, C 0.000 }
gfCNCPoint1[448] = {X 441.0276, Y 20.1645, Z -1.3333, A 0.000, B 0.000, C 0.000 }
gfCNCPoint1[449] = {X 440.8579, Y 20.9682, Z -1.3333, A 0.000, B 0.000, C 0.000 }
gfCNCPoint1[450] = {X 440.8512, Y 21.7896, Z -1.3333, A 0.000, B 0.000, C 0.000 }
gfCNCPoint1[451] = {X 441.0080, Y 22.5960, Z -1.3333, A 0.000, B 0.000, C 0.000 }
gfCNCPoint1[452] = {X 441.3527, Y 22.7079, Z -1.3333, A 0.000, B 0.000, C 0.000 }
gfCNCPoint1[453] = {X 441.7101, Y 22.7678, Z -1.3333, A 0.000, B 0.000, C 0.000 }
gfCNCPoint1[454] = {X 443.0506, Y 22.8566, Z -1.3333, A 0.000, B 0.000, C 0.000 }
gfCNCPoint1[455] = {X 444.3938, Y 22.8760, Z -1.3333, A 0.000, B 0.000, C 0.000 }
gfCNCPoint1[456] = {X 445.9273, Y 22.8760, Z -1.3333, A 0.000, B 0.000, C 0.000 }
gfCNCPoint1[457] = {X 449.9121, Y 22.5274, Z -1.3333, A 0.000, B 0.000, C 0.000 }
gfCNCPoint1[458] = {X 441.9425, Y 22.6074, Z -1.3333, A 0.000, B 0.000, C 0.000 }
gfCNCPoint1[459] = {X 445.9273, Y 22.9560, Z -1.3333, A 0.000, B 0.000, C 0.000 }
gfCNCPoint1[460] = {X 450.5184, Y 22.9560, Z -1.3333, A 0.000, B 0.000, C 0.000 }
gfCNCPoint1[461] = {X 450.5199, Y 19.3810, Z -1.3333, A 0.000, B 0.000, C 0.000 }
gfCNCPoint1[462] = {X 444.0367, Y 19.3804, Z -1.3333, A 0.000, B 0.000, C 0.000 }
gfCNCPoint1[463] = {X 443.3442, Y 19.3967, Z -1.3333, A 0.000, B 0.000, C 0.000 }
gfCNCPoint1[464] = {X 442.3276, Y 19.4902, Z -1.3333, A 0.000, B 0.000, C 0.000 }
gfCNCPoint1[465] = {X 441.3387, Y 19.7440, Z -1.3333, A 0.000, B 0.000, C 0.000 }
gfCNCPoint1[466] = {X 441.0980, Y 19.8962, Z -1.3333, A 0.000, B 0.000, C 0.000 }
gfCNCPoint1[467] = {X 440.9514, Y 20.1402, Z -1.3333, A 0.000, B 0.000, C 0.000 }
gfCNCPoint1[468] = {X 440.7770, Y 20.9722, Z -1.3333, A 0.000, B 0.000, C 0.000 }
gfCNCPoint1[469] = {X 440.7740, Y 21.8222, Z -1.3333, A 0.000, B 0.000, C 0.000 }
gfCNCPoint1[470] = {X 440.9425, Y 22.6553, Z -1.3333, A 0.000, B 0.000, C 0.000 }
gfCNCPoint1[471] = {X 441.3151, Y 22.7810, Z -1.3333, A 0.000, B 0.000, C 0.000 }
gfCNCPoint1[472] = {X 441.7028, Y 22.8475, Z -1.3333, A 0.000, B 0.000, C 0.000 }
gfCNCPoint1[473] = {X 443.0471, Y 22.9365, Z -1.3333, A 0.000, B 0.000, C 0.000 }
gfCNCPoint1[474] = {X 444.3942, Y 22.9560, Z -1.3333, A 0.000, B 0.000, C 0.000 }
gfCNCPoint1[475] = {X 445.9273, Y 22.9560, Z -1.3333, A 0.000, B 0.000, C 0.000 }
gfCNCPoint1[476] = {X 449.9121, Y 22.6074, Z -1.3333, A 0.000, B 0.000, C 0.000 }
gfCNCPoint1[477] = {X 449.9121, Y 22.6074, Z 1.6667, A 0.000, B 0.000, C 0.000 }
gfCNCPoint1[478] = {X 449.9121, Y 22.6074, Z 11.0000, A 0.000, B 0.000, C 0.000 }
gfCNCPoint1[479] = {X 507.6820, Y 107.6949, Z 11.0000, A 0.000, B 0.000, C 0.000 }
gfCNCPoint1[480] = {X 507.6820, Y 107.6949, Z 1.6667, A 0.000, B 0.000, C 0.000 }
gfCNCPoint1[481] = {X 507.6820, Y 107.6949, Z -1.3333, A 0.000, B 0.000, C 0.000 }
gfCNCPoint1[482] = {X 507.6820, Y 71.2949, Z -1.3333, A 0.000, B 0.000, C 0.000 }
gfCNCPoint1[483] = {X 509.5499, Y 71.2949, Z -1.3333, A 0.000, B 0.000, C 0.000 }
gfCNCPoint1[484] = {X 509.0277, Y 71.0690, Z -1.3333, A 0.000, B 0.000, C 0.000 }
gfCNCPoint1[485] = {X 508.5105, Y 70.8320, Z -1.3333, A 0.000, B 0.000, C 0.000 }
gfCNCPoint1[486] = {X 507.1683, Y 71.0983, Z -1.3333, A 0.000, B 0.000, C 0.000 }
gfCNCPoint1[487] = {X 505.8141, Y 71.2949, Z -1.3333, A 0.000, B 0.000, C 0.000 }
gfCNCPoint1[488] = {X 507.6820, Y 71.2949, Z -1.3333, A 0.000, B 0.000, C 0.000 }
gfCNCPoint1[489] = {X 507.6820, Y 73.6949, Z -1.3333, A 0.000, B 0.000, C 0.000 }
gfCNCPoint1[490] = {X 551.2531, Y 73.6949, Z -1.3333, A 0.000, B 0.000, C 0.000 }
gfCNCPoint1[491] = {X 549.1231, Y 72.7702, Z -1.3333, A 0.000, B 0.000, C 0.000 }
gfCNCPoint1[492] = {X 547.0688, Y 71.6877, Z -1.3333, A 0.000, B 0.000, C 0.000 }
gfCNCPoint1[493] = {X 545.1019, Y 70.4535, Z -1.3333, A 0.000, B 0.000, C 0.000 }
gfCNCPoint1[494] = {X 543.2335, Y 69.0746, Z -1.3333, A 0.000, B 0.000, C 0.000 }
gfCNCPoint1[495] = {X 529.7643, Y 69.0750, Z -1.3333, A 0.000, B 0.000, C 0.000 }
gfCNCPoint1[496] = {X 527.5566, Y 69.8771, Z -1.3333, A 0.000, B 0.000, C 0.000 }
gfCNCPoint1[497] = {X 525.2816, Y 70.4617, Z -1.3333, A 0.000, B 0.000, C 0.000 }
gfCNCPoint1[498] = {X 522.9607, Y 70.8234, Z -1.3333, A 0.000, B 0.000, C 0.000 }
gfCNCPoint1[499] = {X 520.6157, Y 70.9587, Z -1.3333, A 0.000, B 0.000, C 0.000 }
gfCNCPoint1[500] = {X 519.7998, Y 70.9591, Z -1.3333, A 0.000, B 0.000, C 0.000 }
gfCNCPoint1[501] = {X 517.4110, Y 70.8403, Z -1.3333, A 0.000, B 0.000, C 0.000 }
gfCNCPoint1[502] = {X 515.0457, Y 70.4852, Z -1.3333, A 0.000, B 0.000, C 0.000 }
gfCNCPoint1[503] = {X 512.7274, Y 69.8971, Z -1.3333, A 0.000, B 0.000, C 0.000 }
gfCNCPoint1[504] = {X 510.4789, Y 69.0820, Z -1.3333, A 0.000, B 0.000, C 0.000 }
gfCNCPoint1[505] = {X 509.6264, Y 68.7045, Z -1.3333, A 0.000, B 0.000, C 0.000 }
gfCNCPoint1[506] = {X 508.7892, Y 68.2944, Z -1.3333, A 0.000, B 0.000, C 0.000 }
gfCNCPoint1[507] = {X 507.1706, Y 68.6592, Z -1.3333, A 0.000, B 0.000, C 0.000 }
gfCNCPoint1[508] = {X 505.5308, Y 68.9117, Z -1.3333, A 0.000, B 0.000, C 0.000 }
gfCNCPoint1[509] = {X 504.1121, Y 69.0379, Z -1.3333, A 0.000, B 0.000, C 0.000 }
gfCNCPoint1[510] = {X 502.6885, Y 69.0800, Z -1.3333, A 0.000, B 0.000, C 0.000 }
gfCNCPoint1[511] = {X 502.0391, Y 69.0800, Z -1.3333, A 0.000, B 0.000, C 0.000 }
gfCNCPoint1[512] = {X 501.1770, Y 71.1331, Z -1.3333, A 0.000, B 0.000, C 0.000 }
gfCNCPoint1[513] = {X 500.1593, Y 73.1137, Z -1.3333, A 0.000, B 0.000, C 0.000 }
gfCNCPoint1[514] = {X 500.1594, Y 73.6949, Z -1.3333, A 0.000, B 0.000, C 0.000 }
gfCNCPoint1[515] = {X 507.6820, Y 73.6949, Z -1.3333, A 0.000, B 0.000, C 0.000 }
gfCNCPoint1[516] = {X 507.6820, Y 76.0949, Z -1.3333, A 0.000, B 0.000, C 0.000 }
gfCNCPoint1[517] = {X 576.0965, Y 76.0949, Z -1.3333, A 0.000, B 0.000, C 0.000 }
gfCNCPoint1[518] = {X 576.0965, Y 72.8901, Z -1.3333, A 0.000, B 0.000, C 0.000 }
gfCNCPoint1[519] = {X 575.7178, Y 72.8147, Z -1.3333, A 0.000, B 0.000, C 0.000 }
gfCNCPoint1[520] = {X 575.3401, Y 72.7341, Z -1.3333, A 0.000, B 0.000, C 0.000 }
gfCNCPoint1[521] = {X 573.3201, Y 73.1034, Z -1.3333, A 0.000, B 0.000, C 0.000 }
gfCNCPoint1[522] = {X 571.2786, Y 73.3258, Z -1.3333, A 0.000, B 0.000, C 0.000 }
gfCNCPoint1[523] = {X 569.2264, Y 73.4000, Z -1.3333, A 0.000, B 0.000, C 0.000 }
gfCNCPoint1[524] = {X 562.4443, Y 73.4000, Z -1.3333, A 0.000, B 0.000, C 0.000 }
gfCNCPoint1[525] = {X 560.3341, Y 73.3215, Z -1.3333, A 0.000, B 0.000, C 0.000 }
gfCNCPoint1[526] = {X 558.2355, Y 73.0864, Z -1.3333, A 0.000, B 0.000, C 0.000 }
gfCNCPoint1[527] = {X 556.1602, Y 72.6960, Z -1.3333, A 0.000, B 0.000, C 0.000 }
gfCNCPoint1[528] = {X 554.1197, Y 72.1525, Z -1.3333, A 0.000, B 0.000, C 0.000 }
gfCNCPoint1[529] = {X 552.1251, Y 71.4589, Z -1.3333, A 0.000, B 0.000, C 0.000 }
gfCNCPoint1[530] = {X 549.9755, Y 70.5165, Z -1.3333, A 0.000, B 0.000, C 0.000 }
gfCNCPoint1[531] = {X 547.9111, Y 69.3997, Z -1.3333, A 0.000, B 0.000, C 0.000 }
gfCNCPoint1[532] = {X 545.9459, Y 68.1163, Z -1.3333, A 0.000, B 0.000, C 0.000 }
gfCNCPoint1[533] = {X 544.0934, Y 66.6750, Z -1.3333, A 0.000, B 0.000, C 0.000 }
gfCNCPoint1[534] = {X 543.8495, Y 66.6762, Z -1.3333, A 0.000, B 0.000, C 0.000 }
gfCNCPoint1[535] = {X 543.6056, Y 66.6746, Z -1.3333, A 0.000, B 0.000, C 0.000 }
gfCNCPoint1[536] = {X 529.2684, Y 66.6750, Z -1.3333, A 0.000, B 0.000, C 0.000 }
gfCNCPoint1[537] = {X 527.1860, Y 67.4765, Z -1.3333, A 0.000, B 0.000, C 0.000 }
gfCNCPoint1[538] = {X 525.0326, Y 68.0613, Z -1.3333, A 0.000, B 0.000, C 0.000 }
gfCNCPoint1[539] = {X 522.8308, Y 68.4233, Z -1.3333, A 0.000, B 0.000, C 0.000 }
gfCNCPoint1[540] = {X 520.6035, Y 68.5587, Z -1.3333, A 0.000, B 0.000, C 0.000 }
gfCNCPoint1[541] = {X 519.7998, Y 68.5591, Z -1.3333, A 0.000, B 0.000, C 0.000 }
gfCNCPoint1[542] = {X 517.5593, Y 68.4430, Z -1.3333, A 0.000, B 0.000, C 0.000 }
gfCNCPoint1[543] = {X 515.3429, Y 68.0961, Z -1.3333, A 0.000, B 0.000, C 0.000 }
gfCNCPoint1[544] = {X 513.1742, Y 67.5219, Z -1.3333, A 0.000, B 0.000, C 0.000 }
gfCNCPoint1[545] = {X 511.0764, Y 66.7267, Z -1.3333, A 0.000, B 0.000, C 0.000 }
gfCNCPoint1[546] = {X 509.0720, Y 65.7189, Z -1.3333, A 0.000, B 0.000, C 0.000 }
gfCNCPoint1[547] = {X 506.9797, Y 66.2511, Z -1.3333, A 0.000, B 0.000, C 0.000 }
gfCNCPoint1[548] = {X 504.8448, Y 66.5725, Z -1.3333, A 0.000, B 0.000, C 0.000 }
gfCNCPoint1[549] = {X 502.6885, Y 66.6800, Z -1.3333, A 0.000, B 0.000, C 0.000 }
gfCNCPoint1[550] = {X 500.3217, Y 66.6800, Z -1.3333, A 0.000, B 0.000, C 0.000 }
gfCNCPoint1[551] = {X 499.6228, Y 68.6760, Z -1.3333, A 0.000, B 0.000, C 0.000 }
gfCNCPoint1[552] = {X 498.7669, Y 70.6099, Z -1.3333, A 0.000, B 0.000, C 0.000 }
gfCNCPoint1[553] = {X 497.7593, Y 72.4693, Z -1.3333, A 0.000, B 0.000, C 0.000 }
gfCNCPoint1[554] = {X 497.7594, Y 76.0949, Z -1.3333, A 0.000, B 0.000, C 0.000 }
gfCNCPoint1[555] = {X 507.6820, Y 76.0949, Z -1.3333, A 0.000, B 0.000, C 0.000 }
gfCNCPoint1[556] = {X 507.6820, Y 78.4949, Z -1.3333, A 0.000, B 0.000, C 0.000 }
gfCNCPoint1[557] = {X 578.4965, Y 78.4949, Z -1.3333, A 0.000, B 0.000, C 0.000 }
gfCNCPoint1[558] = {X 578.4965, Y 70.8313, Z -1.3333, A 0.000, B 0.000, C 0.000 }
gfCNCPoint1[559] = {X 576.9097, Y 70.5998, Z -1.3333, A 0.000, B 0.000, C 0.000 }
gfCNCPoint1[560] = {X 575.3401, Y 70.2710, Z -1.3333, A 0.000, B 0.000, C 0.000 }
gfCNCPoint1[561] = {X 573.3236, Y 70.6751, Z -1.3333, A 0.000, B 0.000, C 0.000 }
gfCNCPoint1[562] = {X 571.2815, Y 70.9187, Z -1.3333, A 0.000, B 0.000, C 0.000 }
gfCNCPoint1[563] = {X 569.2264, Y 71.0000, Z -1.3333, A 0.000, B 0.000, C 0.000 }
gfCNCPoint1[564] = {X 562.4443, Y 71.0000, Z -1.3333, A 0.000, B 0.000, C 0.000 }
gfCNCPoint1[565] = {X 560.0510, Y 70.8896, Z -1.3333, A 0.000, B 0.000, C 0.000 }
gfCNCPoint1[566] = {X 557.6781, Y 70.5594, Z -1.3333, A 0.000, B 0.000, C 0.000 }
gfCNCPoint1[567] = {X 555.3456, Y 70.0122, Z -1.3333, A 0.000, B 0.000, C 0.000 }
gfCNCPoint1[568] = {X 553.0734, Y 69.2525, Z -1.3333, A 0.000, B 0.000, C 0.000 }
gfCNCPoint1[569] = {X 550.8807, Y 68.2870, Z -1.3333, A 0.000, B 0.000, C 0.000 }
gfCNCPoint1[570] = {X 548.7863, Y 67.1237, Z -1.3333, A 0.000, B 0.000, C 0.000 }
gfCNCPoint1[571] = {X 546.8078, Y 65.7726, Z -1.3333, A 0.000, B 0.000, C 0.000 }
gfCNCPoint1[572] = {X 544.9621, Y 64.2450, Z -1.3333, A 0.000, B 0.000, C 0.000 }
gfCNCPoint1[573] = {X 544.2915, Y 64.2715, Z -1.3333, A 0.000, B 0.000, C 0.000 }
gfCNCPoint1[574] = {X 543.6204, Y 64.2746, Z -1.3333, A 0.000, B 0.000, C 0.000 }
gfCNCPoint1[575] = {X 528.7432, Y 64.2750, Z -1.3333, A 0.000, B 0.000, C 0.000 }
gfCNCPoint1[576] = {X 526.7915, Y 65.0766, Z -1.3333, A 0.000, B 0.000, C 0.000 }
gfCNCPoint1[577] = {X 524.7644, Y 65.6619, Z -1.3333, A 0.000, B 0.000, C 0.000 }
gfCNCPoint1[578] = {X 522.6857, Y 66.0241, Z -1.3333, A 0.000, B 0.000, C 0.000 }
gfCNCPoint1[579] = {X 520.5801, Y 66.1588, Z -1.3333, A 0.000, B 0.000, C 0.000 }
gfCNCPoint1[580] = {X 519.7998, Y 66.1591, Z -1.3333, A 0.000, B 0.000, C 0.000 }
gfCNCPoint1[581] = {X 517.9641, Y 66.0715, Z -1.3333, A 0.000, B 0.000, C 0.000 }
gfCNCPoint1[582] = {X 516.1450, Y 65.8096, Z -1.3333, A 0.000, B 0.000, C 0.000 }
gfCNCPoint1[583] = {X 514.3592, Y 65.3756, Z -1.3333, A 0.000, B 0.000, C 0.000 }
gfCNCPoint1[584] = {X 512.6228, Y 64.7735, Z -1.3333, A 0.000, B 0.000, C 0.000 }
gfCNCPoint1[585] = {X 510.9516, Y 64.0089, Z -1.3333, A 0.000, B 0.000, C 0.000 }
gfCNCPoint1[586] = {X 509.3609, Y 63.0886, Z -1.3333, A 0.000, B 0.000, C 0.000 }
gfCNCPoint1[587] = {X 507.7389, Y 63.6068, Z -1.3333, A 0.000, B 0.000, C 0.000 }
gfCNCPoint1[588] = {X 506.0774, Y 63.9798, Z -1.3333, A 0.000, B 0.000, C 0.000 }
gfCNCPoint1[589] = {X 504.3896, Y 64.2048, Z -1.3333, A 0.000, B 0.000, C 0.000 }
gfCNCPoint1[590] = {X 502.6885, Y 64.2800, Z -1.3333, A 0.000, B 0.000, C 0.000 }
gfCNCPoint1[591] = {X 498.4791, Y 64.2800, Z -1.3333, A 0.000, B 0.000, C 0.000 }
gfCNCPoint1[592] = {X 497.9415, Y 66.2508, Z -1.3333, A 0.000, B 0.000, C 0.000 }
gfCNCPoint1[593] = {X 497.2387, Y 68.1690, Z -1.3333, A 0.000, B 0.000, C 0.000 }
gfCNCPoint1[594] = {X 496.3760, Y 70.0208, Z -1.3333, A 0.000, B 0.000, C 0.000 }
gfCNCPoint1[595] = {X 495.3593, Y 71.7927, Z -1.3333, A 0.000, B 0.000, C 0.000 }
gfCNCPoint1[596] = {X 495.3594, Y 78.4949, Z -1.3333, A 0.000, B 0.000, C 0.000 }
gfCNCPoint1[597] = {X 507.6820, Y 78.4949, Z -1.3333, A 0.000, B 0.000, C 0.000 }
gfCNCPoint1[598] = {X 507.6820, Y 80.8949, Z -1.3333, A 0.000, B 0.000, C 0.000 }
gfCNCPoint1[599] = {X 580.8965, Y 80.8949, Z -1.3333, A 0.000, B 0.000, C 0.000 }
gfCNCPoint1[600] = {X 580.8965, Y 68.5934, Z -1.3333, A 0.000, B 0.000, C 0.000 }
gfCNCPoint1[601] = {X 579.0251, Y 68.4747, Z -1.3333, A 0.000, B 0.000, C 0.000 }
gfCNCPoint1[602] = {X 577.1691, Y 68.2078, Z -1.3333, A 0.000, B 0.000, C 0.000 }
gfCNCPoint1[603] = {X 575.3401, Y 67.7943, Z -1.3333, A 0.000, B 0.000, C 0.000 }
gfCNCPoint1[604] = {X 573.3283, Y 68.2408, Z -1.3333, A 0.000, B 0.000, C 0.000 }
gfCNCPoint1[605] = {X 571.2852, Y 68.5100, Z -1.3333, A 0.000, B 0.000, C 0.000 }
gfCNCPoint1[606] = {X 569.2264, Y 68.6000, Z -1.3333, A 0.000, B 0.000, C 0.000 }
gfCNCPoint1[607] = {X 562.4443, Y 68.6000, Z -1.3333, A 0.000, B 0.000, C 0.000 }
gfCNCPoint1[608] = {X 560.1441, Y 68.4876, Z -1.3333, A 0.000, B 0.000, C 0.000 }
gfCNCPoint1[609] = {X 557.8658, Y 68.1516, Z -1.3333, A 0.000, B 0.000, C 0.000 }
gfCNCPoint1[610] = {X 555.6311, Y 67.5951, Z -1.3333, A 0.000, B 0.000, C 0.000 }
gfCNCPoint1[611] = {X 553.4613, Y 66.8235, Z -1.3333, A 0.000, B 0.000, C 0.000 }
gfCNCPoint1[612] = {X 551.3771, Y 65.8441, Z -1.3333, A 0.000, B 0.000, C 0.000 }
gfCNCPoint1[613] = {X 549.3982, Y 64.6662, Z -1.3333, A 0.000, B 0.000, C 0.000 }
gfCNCPoint1[614] = {X 547.5435, Y 63.3010, Z -1.3333, A 0.000, B 0.000, C 0.000 }
gfCNCPoint1[615] = {X 545.8307, Y 61.7615, Z -1.3333, A 0.000, B 0.000, C 0.000 }
gfCNCPoint1[616] = {X 544.7353, Y 61.8538, Z -1.3333, A 0.000, B 0.000, C 0.000 }
gfCNCPoint1[617] = {X 543.6362, Y 61.8746, Z -1.3333, A 0.000, B 0.000, C 0.000 }
gfCNCPoint1[618] = {X 528.1827, Y 61.8750, Z -1.3333, A 0.000, B 0.000, C 0.000 }
gfCNCPoint1[619] = {X 526.3741, Y 62.6756, Z -1.3333, A 0.000, B 0.000, C 0.000 }
gfCNCPoint1[620] = {X 524.4849, Y 63.2611, Z -1.3333, A 0.000, B 0.000, C 0.000 }
gfCNCPoint1[621] = {X 522.5406, Y 63.6239, Z -1.3333, A 0.000, B 0.000, C 0.000 }
gfCNCPoint1[622] = {X 520.5674, Y 63.7588, Z -1.3333, A 0.000, B 0.000, C 0.000 }
gfCNCPoint1[623] = {X 519.7998, Y 63.7591, Z -1.3333, A 0.000, B 0.000, C 0.000 }
gfCNCPoint1[624] = {X 517.9902, Y 63.6618, Z -1.3333, A 0.000, B 0.000, C 0.000 }
gfCNCPoint1[625] = {X 516.2015, Y 63.3711, Z -1.3333, A 0.000, B 0.000, C 0.000 }
gfCNCPoint1[626] = {X 514.4543, Y 62.8904, Z -1.3333, A 0.000, B 0.000, C 0.000 }
gfCNCPoint1[627] = {X 512.7687, Y 62.2251, Z -1.3333, A 0.000, B 0.000, C 0.000 }
gfCNCPoint1[628] = {X 511.1641, Y 61.3829, Z -1.3333, A 0.000, B 0.000, C 0.000 }
gfCNCPoint1[629] = {X 509.6590, Y 60.3735, Z -1.3333, A 0.000, B 0.000, C 0.000 }
gfCNCPoint1[630] = {X 507.9866, Y 61.0270, Z -1.3333, A 0.000, B 0.000, C 0.000 }
gfCNCPoint1[631] = {X 506.2542, Y 61.4991, Z -1.3333, A 0.000, B 0.000, C 0.000 }
gfCNCPoint1[632] = {X 504.4815, Y 61.7845, Z -1.3333, A 0.000, B 0.000, C 0.000 }
gfCNCPoint1[633] = {X 502.6885, Y 61.8800, Z -1.3333, A 0.000, B 0.000, C 0.000 }
gfCNCPoint1[634] = {X 496.4789, Y 61.8800, Z -1.3333, A 0.000, B 0.000, C 0.000 }
gfCNCPoint1[635] = {X 496.1191, Y 63.8335, Z -1.3333, A 0.000, B 0.000, C 0.000 }
gfCNCPoint1[636] = {X 495.5820, Y 65.7460, Z -1.3333, A 0.000, B 0.000, C 0.000 }
gfCNCPoint1[637] = {X 494.8722, Y 67.6012, Z -1.3333, A 0.000, B 0.000, C 0.000 }
gfCNCPoint1[638] = {X 493.9955, Y 69.3837, Z -1.3333, A 0.000, B 0.000, C 0.000 }
gfCNCPoint1[639] = {X 492.9593, Y 71.0784, Z -1.3333, A 0.000, B 0.000, C 0.000 }
gfCNCPoint1[640] = {X 492.9595, Y 80.8949, Z -1.3333, A 0.000, B 0.000, C 0.000 }
gfCNCPoint1[641] = {X 507.6820, Y 80.8949, Z -1.3333, A 0.000, B 0.000, C 0.000 }
gfCNCPoint1[642] = {X 507.6820, Y 83.2949, Z -1.3333, A 0.000, B 0.000, C 0.000 }
gfCNCPoint1[643] = {X 583.2965, Y 83.2949, Z -1.3333, A 0.000, B 0.000, C 0.000 }
gfCNCPoint1[644] = {X 583.2965, Y 66.1198, Z -1.3333, A 0.000, B 0.000, C 0.000 }
gfCNCPoint1[645] = {X 581.2871, Y 66.1993, Z -1.3333, A 0.000, B 0.000, C 0.000 }
gfCNCPoint1[646] = {X 579.2793, Y 66.0882, Z -1.3333, A 0.000, B 0.000, C 0.000 }
gfCNCPoint1[647] = {X 577.2910, Y 65.7873, Z -1.3333, A 0.000, B 0.000, C 0.000 }
gfCNCPoint1[648] = {X 575.3401, Y 65.2993, Z -1.3333, A 0.000, B 0.000, C 0.000 }
gfCNCPoint1[649] = {X 573.3348, Y 65.7981, Z -1.3333, A 0.000, B 0.000, C 0.000 }
gfCNCPoint1[650] = {X 571.2904, Y 66.0993, Z -1.3333, A 0.000, B 0.000, C 0.000 }
gfCNCPoint1[651] = {X 569.2264, Y 66.2000, Z -1.3333, A 0.000, B 0.000, C 0.000 }
gfCNCPoint1[652] = {X 562.4443, Y 66.2000, Z -1.3333, A 0.000, B 0.000, C 0.000 }
gfCNCPoint1[653] = {X 560.2301, Y 66.0841, Z -1.3333, A 0.000, B 0.000, C 0.000 }
gfCNCPoint1[654] = {X 558.0402, Y 65.7375, Z -1.3333, A 0.000, B 0.000, C 0.000 }
gfCNCPoint1[655] = {X 555.8984, Y 65.1641, Z -1.3333, A 0.000, B 0.000, C 0.000 }
gfCNCPoint1[656] = {X 553.8282, Y 64.3701, Z -1.3333, A 0.000, B 0.000, C 0.000 }
gfCNCPoint1[657] = {X 551.8522, Y 63.3643, Z -1.3333, A 0.000, B 0.000, C 0.000 }
gfCNCPoint1[658] = {X 549.9922, Y 62.1576, Z -1.3333, A 0.000, B 0.000, C 0.000 }
gfCNCPoint1[659] = {X 548.2683, Y 60.7633, Z -1.3333, A 0.000, B 0.000, C 0.000 }
gfCNCPoint1[660] = {X 546.6995, Y 59.1965, Z -1.3333, A 0.000, B 0.000, C 0.000 }
gfCNCPoint1[661] = {X 545.1837, Y 59.4162, Z -1.3333, A 0.000, B 0.000, C 0.000 }
gfCNCPoint1[662] = {X 543.6532, Y 59.4746, Z -1.3333, A 0.000, B 0.000, C 0.000 }
gfCNCPoint1[663] = {X 527.5785, Y 59.4751, Z -1.3333, A 0.000, B 0.000, C 0.000 }
gfCNCPoint1[664] = {X 525.9253, Y 60.2742, Z -1.3333, A 0.000, B 0.000, C 0.000 }
gfCNCPoint1[665] = {X 524.1850, Y 60.8601, Z -1.3333, A 0.000, B 0.000, C 0.000 }
gfCNCPoint1[666] = {X 522.3851, Y 61.2236, Z -1.3333, A 0.000, B 0.000, C 0.000 }
gfCNCPoint1[667] = {X 520.5538, Y 61.3588, Z -1.3333, A 0.000, B 0.000, C 0.000 }
gfCNCPoint1[668] = {X 519.7998, Y 61.3591, Z -1.3333, A 0.000, B 0.000, C 0.000 }
gfCNCPoint1[669] = {X 518.0043, Y 61.2474, Z -1.3333, A 0.000, B 0.000, C 0.000 }
gfCNCPoint1[670] = {X 516.2365, Y 60.9138, Z -1.3333, A 0.000, B 0.000, C 0.000 }
gfCNCPoint1[671] = {X 514.5237, Y 60.3637, Z -1.3333, A 0.000, B 0.000, C 0.000 }
gfCNCPoint1[672] = {X 512.8923, Y 59.6054, Z -1.3333, A 0.000, B 0.000, C 0.000 }
gfCNCPoint1[673] = {X 511.3676, Y 58.6507, Z -1.3333, A 0.000, B 0.000, C 0.000 }
gfCNCPoint1[674] = {X 509.9730, Y 57.5142, Z -1.3333, A 0.000, B 0.000, C 0.000 }
gfCNCPoint1[675] = {X 508.6156, Y 58.2113, Z -1.3333, A 0.000, B 0.000, C 0.000 }
gfCNCPoint1[676] = {X 507.1924, Y 58.7617, Z -1.3333, A 0.000, B 0.000, C 0.000 }
gfCNCPoint1[677] = {X 505.7192, Y 59.1593, Z -1.3333, A 0.000, B 0.000, C 0.000 }
gfCNCPoint1[678] = {X 504.2123, Y 59.3996, Z -1.3333, A 0.000, B 0.000, C 0.000 }
gfCNCPoint1[679] = {X 502.6885, Y 59.4800, Z -1.3333, A 0.000, B 0.000, C 0.000 }
gfCNCPoint1[680] = {X 496.2450, Y 59.4800, Z -1.3333, A 0.000, B 0.000, C 0.000 }
gfCNCPoint1[681] = {X 495.2580, Y 59.4463, Z -1.3333, A 0.000, B 0.000, C 0.000 }
gfCNCPoint1[682] = {X 494.2756, Y 59.3454, Z -1.3333, A 0.000, B 0.000, C 0.000 }
gfCNCPoint1[683] = {X 494.1342, Y 61.3008, Z -1.3333, A 0.000, B 0.000, C 0.000 }
gfCNCPoint1[684] = {X 493.7949, Y 63.2317, Z -1.3333, A 0.000, B 0.000, C 0.000 }
gfCNCPoint1[685] = {X 493.2613, Y 65.1182, Z -1.3333, A 0.000, B 0.000, C 0.000 }
gfCNCPoint1[686] = {X 492.5389, Y 66.9407, Z -1.3333, A 0.000, B 0.000, C 0.000 }
gfCNCPoint1[687] = {X 491.6351, Y 68.6805, Z -1.3333, A 0.000, B 0.000, C 0.000 }
gfCNCPoint1[688] = {X 490.5593, Y 70.3194, Z -1.3333, A 0.000, B 0.000, C 0.000 }
gfCNCPoint1[689] = {X 490.5595, Y 83.2949, Z -1.3333, A 0.000, B 0.000, C 0.000 }
gfCNCPoint1[690] = {X 507.6820, Y 83.2949, Z -1.3333, A 0.000, B 0.000, C 0.000 }
gfCNCPoint1[691] = {X 507.6820, Y 85.6949, Z -1.3333, A 0.000, B 0.000, C 0.000 }
gfCNCPoint1[692] = {X 585.6965, Y 85.6949, Z -1.3333, A 0.000, B 0.000, C 0.000 }
gfCNCPoint1[693] = {X 585.6965, Y 63.3150, Z -1.3333, A 0.000, B 0.000, C 0.000 }
gfCNCPoint1[694] = {X 584.3994, Y 63.5678, Z -1.3333, A 0.000, B 0.000, C 0.000 }
gfCNCPoint1[695] = {X 583.0879, Y 63.7289, Z -1.3333, A 0.000, B 0.000, C 0.000 }
gfCNCPoint1[696] = {X 581.1242, Y 63.7971, Z -1.3333, A 0.000, B 0.000, C 0.000 }
gfCNCPoint1[697] = {X 579.1641, Y 63.6600, Z -1.3333, A 0.000, B 0.000, C 0.000 }
gfCNCPoint1[698] = {X 577.2291, Y 63.3191, Z -1.3333, A 0.000, B 0.000, C 0.000 }
gfCNCPoint1[699] = {X 575.3401, Y 62.7781, Z -1.3333, A 0.000, B 0.000, C 0.000 }
gfCNCPoint1[700] = {X 573.3441, Y 63.3435, Z -1.3333, A 0.000, B 0.000, C 0.000 }
gfCNCPoint1[701] = {X 571.2979, Y 63.6855, Z -1.3333, A 0.000, B 0.000, C 0.000 }
gfCNCPoint1[702] = {X 569.2264, Y 63.8000, Z -1.3333, A 0.000, B 0.000, C 0.000 }
gfCNCPoint1[703] = {X 562.4443, Y 63.8000, Z -1.3333, A 0.000, B 0.000, C 0.000 }
gfCNCPoint1[704] = {X 560.5406, Y 63.7034, Z -1.3333, A 0.000, B 0.000, C 0.000 }
gfCNCPoint1[705] = {X 558.6565, Y 63.4145, Z -1.3333, A 0.000, B 0.000, C 0.000 }
gfCNCPoint1[706] = {X 556.8113, Y 62.9363, Z -1.3333, A 0.000, B 0.000, C 0.000 }
gfCNCPoint1[707] = {X 555.0241, Y 62.2737, Z -1.3333, A 0.000, B 0.000, C 0.000 }
gfCNCPoint1[708] = {X 553.3131, Y 61.4335, Z -1.3333, A 0.000, B 0.000, C 0.000 }
gfCNCPoint1[709] = {X 551.6960, Y 60.4244, Z -1.3333, A 0.000, B 0.000, C 0.000 }
gfCNCPoint1[710] = {X 550.1893, Y 59.2568, Z -1.3333, A 0.000, B 0.000, C 0.000 }
gfCNCPoint1[711] = {X 548.8087, Y 57.9426, Z -1.3333, A 0.000, B 0.000, C 0.000 }
gfCNCPoint1[712] = {X 547.5682, Y 56.4953, Z -1.3333, A 0.000, B 0.000, C 0.000 }
gfCNCPoint1[713] = {X 546.2931, Y 56.8301, Z -1.3333, A 0.000, B 0.000, C 0.000 }
gfCNCPoint1[714] = {X 544.9890, Y 57.0239, Z -1.3333, A 0.000, B 0.000, C 0.000 }
gfCNCPoint1[715] = {X 543.6717, Y 57.0746, Z -1.3333, A 0.000, B 0.000, C 0.000 }
gfCNCPoint1[716] = {X 526.9187, Y 57.0751, Z -1.3333, A 0.000, B 0.000, C 0.000 }
gfCNCPoint1[717] = {X 525.4340, Y 57.8735, Z -1.3333, A 0.000, B 0.000, C 0.000 }
gfCNCPoint1[718] = {X 523.8536, Y 58.4603, Z -1.3333, A 0.000, B 0.000, C 0.000 }
gfCNCPoint1[719] = {X 522.2076, Y 58.8245, Z -1.3333, A 0.000, B 0.000, C 0.000 }
gfCNCPoint1[720] = {X 520.5272, Y 58.9590, Z -1.3333, A 0.000, B 0.000, C 0.000 }
gfCNCPoint1[721] = {X 519.7998, Y 58.9591, Z -1.3333, A 0.000, B 0.000, C 0.000 }
gfCNCPoint1[722] = {X 518.2467, Y 58.8589, Z -1.3333, A 0.000, B 0.000, C 0.000 }
gfCNCPoint1[723] = {X 516.7195, Y 58.5598, Z -1.3333, A 0.000, B 0.000, C 0.000 }
gfCNCPoint1[724] = {X 515.2433, Y 58.0668, Z -1.3333, A 0.000, B 0.000, C 0.000 }
gfCNCPoint1[725] = {X 513.8428, Y 57.3882, Z -1.3333, A 0.000, B 0.000, C 0.000 }
gfCNCPoint1[726] = {X 512.5411, Y 56.5351, Z -1.3333, A 0.000, B 0.000, C 0.000 }
gfCNCPoint1[727] = {X 511.3600, Y 55.5218, Z -1.3333, A 0.000, B 0.000, C 0.000 }
gfCNCPoint1[728] = {X 510.3189, Y 54.3650, Z -1.3333, A 0.000, B 0.000, C 0.000 }
gfCNCPoint1[729] = {X 508.9711, Y 55.3177, Z -1.3333, A 0.000, B 0.000, C 0.000 }
gfCNCPoint1[730] = {X 507.5060, Y 56.0778, Z -1.3333, A 0.000, B 0.000, C 0.000 }
gfCNCPoint1[731] = {X 505.9510, Y 56.6311, Z -1.3333, A 0.000, B 0.000, C 0.000 }
gfCNCPoint1[732] = {X 504.3351, Y 56.9672, Z -1.3333, A 0.000, B 0.000, C 0.000 }
gfCNCPoint1[733] = {X 502.6885, Y 57.0800, Z -1.3333, A 0.000, B 0.000, C 0.000 }
gfCNCPoint1[734] = {X 496.2450, Y 57.0800, Z -1.3333, A 0.000, B 0.000, C 0.000 }
gfCNCPoint1[735] = {X 495.4216, Y 57.0519, Z -1.3333, A 0.000, B 0.000, C 0.000 }
gfCNCPoint1[736] = {X 494.6020, Y 56.9677, Z -1.3333, A 0.000, B 0.000, C 0.000 }
gfCNCPoint1[737] = {X 493.1719, Y 56.6826, Z -1.3333, A 0.000, B 0.000, C 0.000 }
gfCNCPoint1[738] = {X 491.7866, Y 56.2272, Z -1.3333, A 0.000, B 0.000, C 0.000 }
gfCNCPoint1[739] = {X 491.8566, Y 57.1124, Z -1.3333, A 0.000, B 0.000, C 0.000 }
gfCNCPoint1[740] = {X 491.8800, Y 58.0000, Z -1.3333, A 0.000, B 0.000, C 0.000 }
gfCNCPoint1[741] = {X 491.8794, Y 59.0735, Z -1.3333, A 0.000, B 0.000, C 0.000 }
gfCNCPoint1[742] = {X 491.8781, Y 59.1839, Z -1.3333, A 0.000, B 0.000, C 0.000 }
gfCNCPoint1[743] = {X 491.8762, Y 59.2942, Z -1.3333, A 0.000, B 0.000, C 0.000 }
gfCNCPoint1[744] = {X 491.7363, Y 61.1320, Z -1.3333, A 0.000, B 0.000, C 0.000 }
gfCNCPoint1[745] = {X 491.3969, Y 62.9436, Z -1.3333, A 0.000, B 0.000, C 0.000 }
gfCNCPoint1[746] = {X 490.8620, Y 64.7074, Z -1.3333, A 0.000, B 0.000, C 0.000 }
gfCNCPoint1[747] = {X 490.1380, Y 66.4024, Z -1.3333, A 0.000, B 0.000, C 0.000 }
gfCNCPoint1[748] = {X 489.2335, Y 68.0083, Z -1.3333, A 0.000, B 0.000, C 0.000 }
gfCNCPoint1[749] = {X 488.1593, Y 69.5061, Z -1.3333, A 0.000, B 0.000, C 0.000 }
gfCNCPoint1[750] = {X 488.1595, Y 85.6949, Z -1.3333, A 0.000, B 0.000, C 0.000 }
gfCNCPoint1[751] = {X 507.6820, Y 85.6949, Z -1.3333, A 0.000, B 0.000, C 0.000 }
gfCNCPoint1[752] = {X 507.6820, Y 88.0949, Z -1.3333, A 0.000, B 0.000, C 0.000 }
gfCNCPoint1[753] = {X 588.0965, Y 88.0949, Z -1.3333, A 0.000, B 0.000, C 0.000 }
gfCNCPoint1[754] = {X 588.0965, Y 60.4644, Z -1.3333, A 0.000, B 0.000, C 0.000 }
gfCNCPoint1[755] = {X 587.7998, Y 60.3564, Z -1.3333, A 0.000, B 0.000, C 0.000 }
gfCNCPoint1[756] = {X 587.5052, Y 60.2427, Z -1.3333, A 0.000, B 0.000, C 0.000 }
gfCNCPoint1[757] = {X 586.3438, Y 60.6540, Z -1.3333, A 0.000, B 0.000, C 0.000 }
gfCNCPoint1[758] = {X 585.1548, Y 60.9769, Z -1.3333, A 0.000, B 0.000, C 0.000 }
gfCNCPoint1[759] = {X 583.5152, Y 61.2699, Z -1.3333, A 0.000, B 0.000, C 0.000 }
gfCNCPoint1[760] = {X 581.8543, Y 61.3951, Z -1.3333, A 0.000, B 0.000, C 0.000 }
gfCNCPoint1[761] = {X 580.1892, Y 61.3512, Z -1.3333, A 0.000, B 0.000, C 0.000 }
gfCNCPoint1[762] = {X 578.5372, Y 61.1386, Z -1.3333, A 0.000, B 0.000, C 0.000 }
gfCNCPoint1[763] = {X 576.9153, Y 60.7595, Z -1.3333, A 0.000, B 0.000, C 0.000 }
gfCNCPoint1[764] = {X 575.3401, Y 60.2178, Z -1.3333, A 0.000, B 0.000, C 0.000 }
gfCNCPoint1[765] = {X 573.8611, Y 60.7315, Z -1.3333, A 0.000, B 0.000, C 0.000 }
gfCNCPoint1[766] = {X 572.3399, Y 61.1017, Z -1.3333, A 0.000, B 0.000, C 0.000 }
gfCNCPoint1[767] = {X 570.7903, Y 61.3253, Z -1.3333, A 0.000, B 0.000, C 0.000 }
gfCNCPoint1[768] = {X 569.2264, Y 61.4000, Z -1.3333, A 0.000, B 0.000, C 0.000 }
gfCNCPoint1[769] = {X 562.4443, Y 61.4000, Z -1.3333, A 0.000, B 0.000, C 0.000 }
gfCNCPoint1[770] = {X 560.5827, Y 61.2940, Z -1.3333, A 0.000, B 0.000, C 0.000 }
gfCNCPoint1[771] = {X 558.7452, Y 60.9774, Z -1.3333, A 0.000, B 0.000, C 0.000 }
gfCNCPoint1[772] = {X 556.9555, Y 60.4542, Z -1.3333, A 0.000, B 0.000, C 0.000 }
gfCNCPoint1[773] = {X 555.2367, Y 59.7313, Z -1.3333, A 0.000, B 0.000, C 0.000 }
gfCNCPoint1[774] = {X 553.6111, Y 58.8179, Z -1.3333, A 0.000, B 0.000, C 0.000 }
gfCNCPoint1[775] = {X 552.0997, Y 57.7260, Z -1.3333, A 0.000, B 0.000, C 0.000 }
gfCNCPoint1[776] = {X 550.7220, Y 56.4695, Z -1.3333, A 0.000, B 0.000, C 0.000 }
gfCNCPoint1[777] = {X 549.4959, Y 55.0647, Z -1.3333, A 0.000, B 0.000, C 0.000 }
gfCNCPoint1[778] = {X 548.4371, Y 53.5299, Z -1.3333, A 0.000, B 0.000, C 0.000 }
gfCNCPoint1[779] = {X 547.3154, Y 54.0413, Z -1.3333, A 0.000, B 0.000, C 0.000 }
gfCNCPoint1[780] = {X 546.1379, Y 54.4061, Z -1.3333, A 0.000, B 0.000, C 0.000 }
gfCNCPoint1[781] = {X 544.9235, Y 54.6183, Z -1.3333, A 0.000, B 0.000, C 0.000 }
gfCNCPoint1[782] = {X 543.6921, Y 54.6746, Z -1.3333, A 0.000, B 0.000, C 0.000 }
gfCNCPoint1[783] = {X 526.1842, Y 54.6751, Z -1.3333, A 0.000, B 0.000, C 0.000 }
gfCNCPoint1[784] = {X 524.8904, Y 55.4719, Z -1.3333, A 0.000, B 0.000, C 0.000 }
gfCNCPoint1[785] = {X 523.4893, Y 56.0599, Z -1.3333, A 0.000, B 0.000, C 0.000 }
gfCNCPoint1[786] = {X 522.0144, Y 56.4252, Z -1.3333, A 0.000, B 0.000, C 0.000 }
gfCNCPoint1[787] = {X 520.5008, Y 56.5591, Z -1.3333, A 0.000, B 0.000, C 0.000 }
gfCNCPoint1[788] = {X 519.7998, Y 56.5591, Z -1.3333, A 0.000, B 0.000, C 0.000 }
gfCNCPoint1[789] = {X 518.3493, Y 56.4498, Z -1.3333, A 0.000, B 0.000, C 0.000 }
gfCNCPoint1[790] = {X 516.9316, Y 56.1244, Z -1.3333, A 0.000, B 0.000, C 0.000 }
gfCNCPoint1[791] = {X 515.5787, Y 55.5903, Z -1.3333, A 0.000, B 0.000, C 0.000 }
gfCNCPoint1[792] = {X 514.3210, Y 54.8595, Z -1.3333, A 0.000, B 0.000, C 0.000 }
gfCNCPoint1[793] = {X 513.1871, Y 53.9484, Z -1.3333, A 0.000, B 0.000, C 0.000 }
gfCNCPoint1[794] = {X 512.2025, Y 52.8778, Z -1.3333, A 0.000, B 0.000, C 0.000 }
gfCNCPoint1[795] = {X 511.3855, Y 51.6648, Z -1.3333, A 0.000, B 0.000, C 0.000 }
gfCNCPoint1[796] = {X 510.7606, Y 50.3426, Z -1.3333, A 0.000, B 0.000, C 0.000 }
gfCNCPoint1[797] = {X 509.8636, Y 51.4977, Z -1.3333, A 0.000, B 0.000, C 0.000 }
gfCNCPoint1[798] = {X 508.8029, Y 52.5044, Z -1.3333, A 0.000, B 0.000, C 0.000 }
gfCNCPoint1[799] = {X 507.7229, Y 53.2678, Z -1.3333, A 0.000, B 0.000, C 0.000 }
gfCNCPoint1[800] = {X 506.5489, Y 53.8769, Z -1.3333, A 0.000, B 0.000, C 0.000 }
gfCNCPoint1[801] = {X 505.3028, Y 54.3203, Z -1.3333, A 0.000, B 0.000, C 0.000 }
gfCNCPoint1[802] = {X 504.0080, Y 54.5896, Z -1.3333, A 0.000, B 0.000, C 0.000 }
gfCNCPoint1[803] = {X 502.6885, Y 54.6800, Z -1.3333, A 0.000, B 0.000, C 0.000 }
gfCNCPoint1[804] = {X 496.2450, Y 54.6800, Z -1.3333, A 0.000, B 0.000, C 0.000 }
gfCNCPoint1[805] = {X 495.0285, Y 54.6033, Z -1.3333, A 0.000, B 0.000, C 0.000 }
gfCNCPoint1[806] = {X 493.8313, Y 54.3742, Z -1.3333, A 0.000, B 0.000, C 0.000 }
gfCNCPoint1[807] = {X 492.6724, Y 53.9966, Z -1.3333, A 0.000, B 0.000, C 0.000 }
gfCNCPoint1[808] = {X 491.4451, Y 53.4062, Z -1.3333, A 0.000, B 0.000, C 0.000 }
gfCNCPoint1[809] = {X 490.3129, Y 52.6493, Z -1.3333, A 0.000, B 0.000, C 0.000 }
gfCNCPoint1[810] = {X 489.2980, Y 51.7410, Z -1.3333, A 0.000, B 0.000, C 0.000 }
gfCNCPoint1[811] = {X 488.8683, Y 52.1573, Z -1.3333, A 0.000, B 0.000, C 0.000 }
gfCNCPoint1[812] = {X 488.4137, Y 52.5463, Z -1.3333, A 0.000, B 0.000, C 0.000 }
gfCNCPoint1[813] = {X 488.8649, Y 53.8245, Z -1.3333, A 0.000, B 0.000, C 0.000 }
gfCNCPoint1[814] = {X 489.1946, Y 55.1393, Z -1.3333, A 0.000, B 0.000, C 0.000 }
gfCNCPoint1[815] = {X 489.3999, Y 56.4792, Z -1.3333, A 0.000, B 0.000, C 0.000 }
gfCNCPoint1[816] = {X 489.4600, Y 57.2386, Z -1.3333, A 0.000, B 0.000, C 0.000 }
gfCNCPoint1[817] = {X 489.4800, Y 58.0000, Z -1.3333, A 0.000, B 0.000, C 0.000 }
gfCNCPoint1[818] = {X 489.4795, Y 59.0537, Z -1.3333, A 0.000, B 0.000, C 0.000 }
gfCNCPoint1[819] = {X 489.3595, Y 60.7980, Z -1.3333, A 0.000, B 0.000, C 0.000 }
gfCNCPoint1[820] = {X 489.0302, Y 62.5151, Z -1.3333, A 0.000, B 0.000, C 0.000 }
gfCNCPoint1[821] = {X 488.4963, Y 64.1800, Z -1.3333, A 0.000, B 0.000, C 0.000 }
gfCNCPoint1[822] = {X 487.7656, Y 65.7685, Z -1.3333, A 0.000, B 0.000, C 0.000 }
gfCNCPoint1[823] = {X 486.8488, Y 67.2573, Z -1.3333, A 0.000, B 0.000, C 0.000 }
gfCNCPoint1[824] = {X 485.7593, Y 68.6247, Z -1.3333, A 0.000, B 0.000, C 0.000 }
gfCNCPoint1[825] = {X 485.7595, Y 87.3801, Z -1.3333, A 0.000, B 0.000, C 0.000 }
gfCNCPoint1[826] = {X 486.0673, Y 87.7326, Z -1.3333, A 0.000, B 0.000, C 0.000 }
gfCNCPoint1[827] = {X 486.3634, Y 88.0949, Z -1.3333, A 0.000, B 0.000, C 0.000 }
gfCNCPoint1[828] = {X 507.6820, Y 88.0949, Z -1.3333, A 0.000, B 0.000, C 0.000 }
gfCNCPoint1[829] = {X 507.6820, Y 90.4949, Z -1.3333, A 0.000, B 0.000, C 0.000 }
gfCNCPoint1[830] = {X 590.4965, Y 90.4949, Z -1.3333, A 0.000, B 0.000, C 0.000 }
gfCNCPoint1[831] = {X 590.4965, Y 58.6615, Z -1.3333, A 0.000, B 0.000, C 0.000 }
gfCNCPoint1[832] = {X 588.9714, Y 58.2279, Z -1.3333, A 0.000, B 0.000, C 0.000 }
gfCNCPoint1[833] = {X 587.5052, Y 57.6246, Z -1.3333, A 0.000, B 0.000, C 0.000 }
gfCNCPoint1[834] = {X 585.8387, Y 58.2956, Z -1.3333, A 0.000, B 0.000, C 0.000 }
gfCNCPoint1[835] = {X 584.0999, Y 58.7477, Z -1.3333, A 0.000, B 0.000, C 0.000 }
gfCNCPoint1[836] = {X 582.3176, Y 58.9733, Z -1.3333, A 0.000, B 0.000, C 0.000 }
gfCNCPoint1[837] = {X 580.5210, Y 58.9689, Z -1.3333, A 0.000, B 0.000, C 0.000 }
gfCNCPoint1[838] = {X 578.7398, Y 58.7344, Z -1.3333, A 0.000, B 0.000, C 0.000 }
gfCNCPoint1[839] = {X 577.0034, Y 58.2738, Z -1.3333, A 0.000, B 0.000, C 0.000 }
gfCNCPoint1[840] = {X 575.3401, Y 57.5945, Z -1.3333, A 0.000, B 0.000, C 0.000 }
gfCNCPoint1[841] = {X 573.8813, Y 58.2035, Z -1.3333, A 0.000, B 0.000, C 0.000 }
gfCNCPoint1[842] = {X 572.3630, Y 58.6441, Z -1.3333, A 0.000, B 0.000, C 0.000 }
gfCNCPoint1[843] = {X 570.8048, Y 58.9107, Z -1.3333, A 0.000, B 0.000, C 0.000 }
gfCNCPoint1[844] = {X 569.2264, Y 59.0000, Z -1.3333, A 0.000, B 0.000, C 0.000 }
gfCNCPoint1[845] = {X 562.4443, Y 59.0000, Z -1.3333, A 0.000, B 0.000, C 0.000 }
gfCNCPoint1[846] = {X 560.6575, Y 58.8855, Z -1.3333, A 0.000, B 0.000, C 0.000 }
gfCNCPoint1[847] = {X 558.9000, Y 58.5439, Z -1.3333, A 0.000, B 0.000, C 0.000 }
gfCNCPoint1[848] = {X 557.2004, Y 57.9808, Z -1.3333, A 0.000, B 0.000, C 0.000 }
gfCNCPoint1[849] = {X 555.5866, Y 57.2054, Z -1.3333, A 0.000, B 0.000, C 0.000 }
gfCNCPoint1[850] = {X 554.0849, Y 56.2303, Z -1.3333, A 0.000, B 0.000, C 0.000 }
gfCNCPoint1[851] = {X 552.7200, Y 55.0716, Z -1.3333, A 0.000, B 0.000, C 0.000 }
gfCNCPoint1[852] = {X 551.5141, Y 53.7481, Z -1.3333, A 0.000, B 0.000, C 0.000 }
gfCNCPoint1[853] = {X 550.4870, Y 52.2816, Z -1.3333, A 0.000, B 0.000, C 0.000 }
gfCNCPoint1[854] = {X 549.8373, Y 51.0879, Z -1.3333, A 0.000, B 0.000, C 0.000 }
gfCNCPoint1[855] = {X 549.3064, Y 49.8368, Z -1.3333, A 0.000, B 0.000, C 0.000 }
gfCNCPoint1[856] = {X 548.3749, Y 50.7136, Z -1.3333, A 0.000, B 0.000, C 0.000 }
gfCNCPoint1[857] = {X 547.3045, Y 51.4139, Z -1.3333, A 0.000, B 0.000, C 0.000 }
gfCNCPoint1[858] = {X 546.1632, Y 51.9047, Z -1.3333, A 0.000, B 0.000, C 0.000 }
gfCNCPoint1[859] = {X 544.9550, Y 52.1944, Z -1.3333, A 0.000, B 0.000, C 0.000 }
gfCNCPoint1[860] = {X 543.7152, Y 52.2746, Z -1.3333, A 0.000, B 0.000, C 0.000 }
gfCNCPoint1[861] = {X 525.3419, Y 52.2751, Z -1.3333, A 0.000, B 0.000, C 0.000 }
gfCNCPoint1[862] = {X 524.2749, Y 53.0668, Z -1.3333, A 0.000, B 0.000, C 0.000 }
gfCNCPoint1[863] = {X 523.0841, Y 53.6560, Z -1.3333, A 0.000, B 0.000, C 0.000 }
gfCNCPoint1[864] = {X 521.8076, Y 54.0240, Z -1.3333, A 0.000, B 0.000, C 0.000 }
gfCNCPoint1[865] = {X 520.4859, Y 54.1591, Z -1.3333, A 0.000, B 0.000, C 0.000 }
gfCNCPoint1[866] = {X 519.7998, Y 54.1591, Z -1.3333, A 0.000, B 0.000, C 0.000 }
gfCNCPoint1[867] = {X 518.5529, Y 54.0515, Z -1.3333, A 0.000, B 0.000, C 0.000 }
gfCNCPoint1[868] = {X 517.3428, Y 53.7320, Z -1.3333, A 0.000, B 0.000, C 0.000 }
gfCNCPoint1[869] = {X 516.2054, Y 53.2099, Z -1.3333, A 0.000, B 0.000, C 0.000 }
gfCNCPoint1[870] = {X 515.1742, Y 52.5007, Z -1.3333, A 0.000, B 0.000, C 0.000 }
gfCNCPoint1[871] = {X 514.2797, Y 51.6254, Z -1.3333, A 0.000, B 0.000, C 0.000 }
gfCNCPoint1[872] = {X 513.5483, Y 50.6098, Z -1.3333, A 0.000, B 0.000, C 0.000 }
gfCNCPoint1[873] = {X 513.0017, Y 49.4839, Z -1.3333, A 0.000, B 0.000, C 0.000 }
gfCNCPoint1[874] = {X 512.7353, Y 48.6374, Z -1.3333, A 0.000, B 0.000, C 0.000 }
gfCNCPoint1[875] = {X 512.5739, Y 47.7649, Z -1.3333, A 0.000, B 0.000, C 0.000 }
gfCNCPoint1[876] = {X 512.5198, Y 46.8791, Z -1.3333, A 0.000, B 0.000, C 0.000 }
gfCNCPoint1[877] = {X 512.5198, Y 39.9011, Z -1.3333, A 0.000, B 0.000, C 0.000 }
gfCNCPoint1[878] = {X 512.5806, Y 38.9618, Z -1.3333, A 0.000, B 0.000, C 0.000 }
gfCNCPoint1[879] = {X 512.7622, Y 38.0382, Z -1.3333, A 0.000, B 0.000, C 0.000 }
gfCNCPoint1[880] = {X 513.0614, Y 37.1457, Z -1.3333, A 0.000, B 0.000, C 0.000 }
gfCNCPoint1[881] = {X 513.5568, Y 36.1562, Z -1.3333, A 0.000, B 0.000, C 0.000 }
gfCNCPoint1[882] = {X 514.1965, Y 35.2533, Z -1.3333, A 0.000, B 0.000, C 0.000 }
gfCNCPoint1[883] = {X 514.9657, Y 34.4578, Z -1.3333, A 0.000, B 0.000, C 0.000 }
gfCNCPoint1[884] = {X 515.8465, Y 33.7880, Z -1.3333, A 0.000, B 0.000, C 0.000 }
gfCNCPoint1[885] = {X 513.2399, Y 29.7574, Z -1.3333, A 0.000, B 0.000, C 0.000 }
gfCNCPoint1[886] = {X 513.5210, Y 29.5811, Z -1.3333, A 0.000, B 0.000, C 0.000 }
gfCNCPoint1[887] = {X 513.8068, Y 29.4125, Z -1.3333, A 0.000, B 0.000, C 0.000 }
gfCNCPoint1[888] = {X 513.8068, Y 27.6757, Z -1.3333, A 0.000, B 0.000, C 0.000 }
gfCNCPoint1[889] = {X 513.5209, Y 27.5007, Z -1.3333, A 0.000, B 0.000, C 0.000 }
gfCNCPoint1[890] = {X 513.2400, Y 27.3179, Z -1.3333, A 0.000, B 0.000, C 0.000 }
gfCNCPoint1[891] = {X 513.2399, Y 29.7574, Z -1.3333, A 0.000, B 0.000, C 0.000 }
gfCNCPoint1[892] = {X 514.5432, Y 31.7727, Z -1.3333, A 0.000, B 0.000, C 0.000 }
gfCNCPoint1[893] = {X 515.3541, Y 31.3023, Z -1.3333, A 0.000, B 0.000, C 0.000 }
gfCNCPoint1[894] = {X 516.2068, Y 30.9126, Z -1.3333, A 0.000, B 0.000, C 0.000 }
gfCNCPoint1[895] = {X 516.2068, Y 26.2046, Z -1.3333, A 0.000, B 0.000, C 0.000 }
gfCNCPoint1[896] = {X 515.3707, Y 25.8038, Z -1.3333, A 0.000, B 0.000, C 0.000 }
gfCNCPoint1[897] = {X 514.5769, Y 25.3248, Z -1.3333, A 0.000, B 0.000, C 0.000 }
gfCNCPoint1[898] = {X 513.5934, Y 24.5694, Z -1.3333, A 0.000, B 0.000, C 0.000 }
gfCNCPoint1[899] = {X 512.7145, Y 23.6945, Z -1.3333, A 0.000, B 0.000, C 0.000 }
gfCNCPoint1[900] = {X 511.9547, Y 22.7145, Z -1.3333, A 0.000, B 0.000, C 0.000 }
gfCNCPoint1[901] = {X 511.3264, Y 21.6453, Z -1.3333, A 0.000, B 0.000, C 0.000 }
gfCNCPoint1[902] = {X 510.8400, Y 20.5046, Z -1.3333, A 0.000, B 0.000, C 0.000 }
gfCNCPoint1[903] = {X 510.8399, Y 36.2373, Z -1.3333, A 0.000, B 0.000, C 0.000 }
gfCNCPoint1[904] = {X 511.4987, Y 34.9217, Z -1.3333, A 0.000, B 0.000, C 0.000 }
gfCNCPoint1[905] = {X 512.3493, Y 33.7211, Z -1.3333, A 0.000, B 0.000, C 0.000 }
gfCNCPoint1[906] = {X 513.3720, Y 32.6633, Z -1.3333, A 0.000, B 0.000, C 0.000 }
gfCNCPoint1[907] = {X 514.5432, Y 31.7727, Z -1.3333, A 0.000, B 0.000, C 0.000 }
gfCNCPoint1[908] = {X 515.8465, Y 33.7880, Z -1.3333, A 0.000, B 0.000, C 0.000 }
gfCNCPoint1[909] = {X 516.7432, Y 33.2939, Z -1.3333, A 0.000, B 0.000, C 0.000 }
gfCNCPoint1[910] = {X 517.7003, Y 32.9304, Z -1.3333, A 0.000, B 0.000, C 0.000 }
gfCNCPoint1[911] = {X 518.6990, Y 32.7048, Z -1.3333, A 0.000, B 0.000, C 0.000 }
gfCNCPoint1[912] = {X 518.6299, Y 32.1290, Z -1.3333, A 0.000, B 0.000, C 0.000 }
gfCNCPoint1[913] = {X 518.6068, Y 31.5495, Z -1.3333, A 0.000, B 0.000, C 0.000 }
gfCNCPoint1[914] = {X 518.6068, Y 24.5714, Z -1.3333, A 0.000, B 0.000, C 0.000 }
gfCNCPoint1[915] = {X 518.6080, Y 24.4373, Z -1.3333, A 0.000, B 0.000, C 0.000 }
gfCNCPoint1[916] = {X 517.3907, Y 24.0938, Z -1.3333, A 0.000, B 0.000, C 0.000 }
gfCNCPoint1[917] = {X 516.2513, Y 23.5448, Z -1.3333, A 0.000, B 0.000, C 0.000 }
gfCNCPoint1[918] = {X 515.2241, Y 22.8069, Z -1.3333, A 0.000, B 0.000, C 0.000 }
gfCNCPoint1[919] = {X 514.3401, Y 21.9023, Z -1.3333, A 0.000, B 0.000, C 0.000 }
gfCNCPoint1[920] = {X 513.6260, Y 20.8583, Z -1.3333, A 0.000, B 0.000, C 0.000 }
gfCNCPoint1[921] = {X 513.1034, Y 19.7065, Z -1.3333, A 0.000, B 0.000, C 0.000 }
gfCNCPoint1[922] = {X 512.7934, Y 18.5137, Z -1.3333, A 0.000, B 0.000, C 0.000 }
gfCNCPoint1[923] = {X 512.6891, Y 17.2857, Z -1.3333, A 0.000, B 0.000, C 0.000 }
gfCNCPoint1[924] = {X 512.6891, Y 10.3077, Z -1.3333, A 0.000, B 0.000, C 0.000 }
gfCNCPoint1[925] = {X 512.7002, Y 9.9058, Z -1.3333, A 0.000, B 0.000, C 0.000 }
gfCNCPoint1[926] = {X 512.7335, Y 9.5051, Z -1.3333, A 0.000, B 0.000, C 0.000 }
gfCNCPoint1[927] = {X 509.4578, Y 9.5051, Z -1.3333, A 0.000, B 0.000, C 0.000 }
gfCNCPoint1[928] = {X 509.7400, Y 10.3732, Z -1.3333, A 0.000, B 0.000, C 0.000 }
gfCNCPoint1[929] = {X 509.9111, Y 11.2698, Z -1.3333, A 0.000, B 0.000, C 0.000 }
gfCNCPoint1[930] = {X 509.9685, Y 12.1807, Z -1.3333, A 0.000, B 0.000, C 0.000 }
gfCNCPoint1[931] = {X 509.9682, Y 13.0462, Z -1.3333, A 0.000, B 0.000, C 0.000 }
gfCNCPoint1[932] = {X 509.8611, Y 14.2240, Z -1.3333, A 0.000, B 0.000, C 0.000 }
gfCNCPoint1[933] = {X 509.5646, Y 15.3690, Z -1.3333, A 0.000, B 0.000, C 0.000 }
gfCNCPoint1[934] = {X 509.0868, Y 16.4509, Z -1.3333, A 0.000, B 0.000, C 0.000 }
gfCNCPoint1[935] = {X 508.4400, Y 17.4411, Z -1.3333, A 0.000, B 0.000, C 0.000 }
gfCNCPoint1[936] = {X 508.4399, Y 39.7457, Z -1.3333, A 0.000, B 0.000, C 0.000 }
gfCNCPoint1[937] = {X 509.0885, Y 40.7392, Z -1.3333, A 0.000, B 0.000, C 0.000 }
gfCNCPoint1[938] = {X 509.5671, Y 41.8249, Z -1.3333, A 0.000, B 0.000, C 0.000 }
gfCNCPoint1[939] = {X 509.8630, Y 42.9739, Z -1.3333, A 0.000, B 0.000, C 0.000 }
gfCNCPoint1[940] = {X 509.9683, Y 44.1558, Z -1.3333, A 0.000, B 0.000, C 0.000 }
gfCNCPoint1[941] = {X 509.9685, Y 45.0000, Z -1.3333, A 0.000, B 0.000, C 0.000 }
gfCNCPoint1[942] = {X 509.8909, Y 46.0603, Z -1.3333, A 0.000, B 0.000, C 0.000 }
gfCNCPoint1[943] = {X 509.6596, Y 47.0980, Z -1.3333, A 0.000, B 0.000, C 0.000 }
gfCNCPoint1[944] = {X 509.2797, Y 48.0910, Z -1.3333, A 0.000, B 0.000, C 0.000 }
gfCNCPoint1[945] = {X 508.7593, Y 49.0180, Z -1.3333, A 0.000, B 0.000, C 0.000 }
gfCNCPoint1[946] = {X 508.0200, Y 49.9571, Z -1.3333, A 0.000, B 0.000, C 0.000 }
gfCNCPoint1[947] = {X 507.1371, Y 50.7626, Z -1.3333, A 0.000, B 0.000, C 0.000 }
gfCNCPoint1[948] = {X 506.1343, Y 51.4129, Z -1.3333, A 0.000, B 0.000, C 0.000 }
gfCNCPoint1[949] = {X 505.0386, Y 51.8902, Z -1.3333, A 0.000, B 0.000, C 0.000 }
gfCNCPoint1[950] = {X 503.8796, Y 52.1819, Z -1.3333, A 0.000, B 0.000, C 0.000 }
gfCNCPoint1[951] = {X 502.6885, Y 52.2800, Z -1.3333, A 0.000, B 0.000, C 0.000 }
gfCNCPoint1[952] = {X 496.2450, Y 52.2800, Z -1.3333, A 0.000, B 0.000, C 0.000 }
gfCNCPoint1[953] = {X 495.0845, Y 52.1869, Z -1.3333, A 0.000, B 0.000, C 0.000 }
gfCNCPoint1[954] = {X 493.9538, Y 51.9100, Z -1.3333, A 0.000, B 0.000, C 0.000 }
gfCNCPoint1[955] = {X 492.8816, Y 51.4564, Z -1.3333, A 0.000, B 0.000, C 0.000 }
gfCNCPoint1[956] = {X 491.8954, Y 50.8377, Z -1.3333, A 0.000, B 0.000, C 0.000 }
gfCNCPoint1[957] = {X 491.0204, Y 50.0697, Z -1.3333, A 0.000, B 0.000, C 0.000 }
gfCNCPoint1[958] = {X 490.2980, Y 49.1989, Z -1.3333, A 0.000, B 0.000, C 0.000 }
gfCNCPoint1[959] = {X 489.7192, Y 48.2267, Z -1.3333, A 0.000, B 0.000, C 0.000 }
gfCNCPoint1[960] = {X 489.2980, Y 47.1766, Z -1.3333, A 0.000, B 0.000, C 0.000 }
gfCNCPoint1[961] = {X 488.8769, Y 48.2267, Z -1.3333, A 0.000, B 0.000, C 0.000 }
gfCNCPoint1[962] = {X 488.2981, Y 49.1989, Z -1.3333, A 0.000, B 0.000, C 0.000 }
gfCNCPoint1[963] = {X 487.5756, Y 50.0697, Z -1.3333, A 0.000, B 0.000, C 0.000 }
gfCNCPoint1[964] = {X 486.8824, Y 50.6978, Z -1.3333, A 0.000, B 0.000, C 0.000 }
gfCNCPoint1[965] = {X 486.1145, Y 51.2318, Z -1.3333, A 0.000, B 0.000, C 0.000 }
gfCNCPoint1[966] = {X 485.2843, Y 51.6629, Z -1.3333, A 0.000, B 0.000, C 0.000 }
gfCNCPoint1[967] = {X 486.0586, Y 53.1385, Z -1.3333, A 0.000, B 0.000, C 0.000 }
gfCNCPoint1[968] = {X 486.6224, Y 54.7067, Z -1.3333, A 0.000, B 0.000, C 0.000 }
gfCNCPoint1[969] = {X 486.9651, Y 56.3375, Z -1.3333, A 0.000, B 0.000, C 0.000 }
gfCNCPoint1[970] = {X 487.0800, Y 58.0000, Z -1.3333, A 0.000, B 0.000, C 0.000 }
gfCNCPoint1[971] = {X 487.0796, Y 59.0339, Z -1.3333, A 0.000, B 0.000, C 0.000 }
gfCNCPoint1[972] = {X 486.9596, Y 60.6354, Z -1.3333, A 0.000, B 0.000, C 0.000 }
gfCNCPoint1[973] = {X 486.6282, Y 62.2069, Z -1.3333, A 0.000, B 0.000, C 0.000 }
gfCNCPoint1[974] = {X 486.0913, Y 63.7205, Z -1.3333, A 0.000, B 0.000, C 0.000 }
gfCNCPoint1[975] = {X 485.3583, Y 65.1495, Z -1.3333, A 0.000, B 0.000, C 0.000 }
gfCNCPoint1[976] = {X 484.4422, Y 66.4687, Z -1.3333, A 0.000, B 0.000, C 0.000 }
gfCNCPoint1[977] = {X 483.3593, Y 67.6547, Z -1.3333, A 0.000, B 0.000, C 0.000 }
gfCNCPoint1[978] = {X 483.3596, Y 88.3512, Z -1.3333, A 0.000, B 0.000, C 0.000 }
gfCNCPoint1[979] = {X 484.3094, Y 89.3716, Z -1.3333, A 0.000, B 0.000, C 0.000 }
gfCNCPoint1[980] = {X 485.1350, Y 90.4949, Z -1.3333, A 0.000, B 0.000, C 0.000 }
gfCNCPoint1[981] = {X 507.6820, Y 90.4949, Z -1.3333, A 0.000, B 0.000, C 0.000 }
gfCNCPoint1[982] = {X 507.6820, Y 92.8949, Z -1.3333, A 0.000, B 0.000, C 0.000 }
gfCNCPoint1[983] = {X 592.8965, Y 92.8949, Z -1.3333, A 0.000, B 0.000, C 0.000 }
gfCNCPoint1[984] = {X 592.8965, Y 56.5812, Z -1.3333, A 0.000, B 0.000, C 0.000 }
gfCNCPoint1[985] = {X 591.4809, Y 56.4128, Z -1.3333, A 0.000, B 0.000, C 0.000 }
gfCNCPoint1[986] = {X 590.0967, Y 56.0720, Z -1.3333, A 0.000, B 0.000, C 0.000 }
gfCNCPoint1[987] = {X 588.7648, Y 55.5640, Z -1.3333, A 0.000, B 0.000, C 0.000 }
gfCNCPoint1[988] = {X 587.5052, Y 54.8965, Z -1.3333, A 0.000, B 0.000, C 0.000 }
gfCNCPoint1[989] = {X 586.9690, Y 55.2051, Z -1.3333, A 0.000, B 0.000, C 0.000 }
gfCNCPoint1[990] = {X 586.4171, Y 55.4846, Z -1.3333, A 0.000, B 0.000, C 0.000 }
gfCNCPoint1[991] = {X 584.8782, Y 56.0830, Z -1.3333, A 0.000, B 0.000, C 0.000 }
gfCNCPoint1[992] = {X 583.2699, Y 56.4570, Z -1.3333, A 0.000, B 0.000, C 0.000 }
gfCNCPoint1[993] = {X 581.6248, Y 56.5987, Z -1.3333, A 0.000, B 0.000, C 0.000 }
gfCNCPoint1[994] = {X 579.9763, Y 56.5055, Z -1.3333, A 0.000, B 0.000, C 0.000 }
gfCNCPoint1[995] = {X 578.3577, Y 56.1792, Z -1.3333, A 0.000, B 0.000, C 0.000 }
gfCNCPoint1[996] = {X 576.8018, Y 55.6263, Z -1.3333, A 0.000, B 0.000, C 0.000 }
gfCNCPoint1[997] = {X 575.3401, Y 54.8581, Z -1.3333, A 0.000, B 0.000, C 0.000 }
gfCNCPoint1[998] = {X 573.9176, Y 55.6091, Z -1.3333, A 0.000, B 0.000, C 0.000 }
gfCNCPoint1[999] = {X 572.4049, Y 56.1560, Z -1.3333, A 0.000, B 0.000, C 0.000 }
gfCNCPoint1[1000] = {X 570.8311, Y 56.4885, Z -1.3333, A 0.000, B 0.000, C 0.000 }
gfCNCPoint1[1001] = {X 569.2264, Y 56.6000, Z -1.3333, A 0.000, B 0.000, C 0.000 }
gfCNCPoint1[1002] = {X 562.4443, Y 56.6000, Z -1.3333, A 0.000, B 0.000, C 0.000 }
gfCNCPoint1[1003] = {X 560.8792, Y 56.4939, Z -1.3333, A 0.000, B 0.000, C 0.000 }
gfCNCPoint1[1004] = {X 559.3427, Y 56.1776, Z -1.3333, A 0.000, B 0.000, C 0.000 }
gfCNCPoint1[1005] = {X 557.8629, Y 55.6569, Z -1.3333, A 0.000, B 0.000, C 0.000 }
gfCNCPoint1[1006] = {X 556.4669, Y 54.9413, Z -1.3333, A 0.000, B 0.000, C 0.000 }
gfCNCPoint1[1007] = {X 555.1802, Y 54.0439, Z -1.3333, A 0.000, B 0.000, C 0.000 }
gfCNCPoint1[1008] = {X 554.0264, Y 52.9811, Z -1.3333, A 0.000, B 0.000, C 0.000 }
gfCNCPoint1[1009] = {X 553.0265, Y 51.7724, Z -1.3333, A 0.000, B 0.000, C 0.000 }
gfCNCPoint1[1010] = {X 552.1988, Y 50.4397, Z -1.3333, A 0.000, B 0.000, C 0.000 }
gfCNCPoint1[1011] = {X 551.5586, Y 49.0076, Z -1.3333, A 0.000, B 0.000, C 0.000 }
gfCNCPoint1[1012] = {X 551.1636, Y 47.7029, Z -1.3333, A 0.000, B 0.000, C 0.000 }
gfCNCPoint1[1013] = {X 550.9244, Y 46.3608, Z -1.3333, A 0.000, B 0.000, C 0.000 }
gfCNCPoint1[1014] = {X 550.8443, Y 45.0000, Z -1.3333, A 0.000, B 0.000, C 0.000 }
gfCNCPoint1[1015] = {X 550.8443, Y 44.0517, Z -1.3333, A 0.000, B 0.000, C 0.000 }
gfCNCPoint1[1016] = {X 550.9574, Y 42.4675, Z -1.3333, A 0.000, B 0.000, C 0.000 }
gfCNCPoint1[1017] = {X 551.2851, Y 40.9135, Z -1.3333, A 0.000, B 0.000, C 0.000 }
gfCNCPoint1[1018] = {X 551.8213, Y 39.4186, Z -1.3333, A 0.000, B 0.000, C 0.000 }
gfCNCPoint1[1019] = {X 549.6228, Y 38.4561, Z -1.3333, A 0.000, B 0.000, C 0.000 }
gfCNCPoint1[1020] = {X 549.7925, Y 38.0834, Z -1.3333, A 0.000, B 0.000, C 0.000 }
gfCNCPoint1[1021] = {X 549.9730, Y 37.7158, Z -1.3333, A 0.000, B 0.000, C 0.000 }
gfCNCPoint1[1022] = {X 549.9730, Y 16.9491, Z -1.3333, A 0.000, B 0.000, C 0.000 }
gfCNCPoint1[1023] = {X 549.8029, Y 17.1989, Z -1.3333, A 0.000, B 0.000, C 0.000 }
gfCNCPoint1[1024] = {X 549.6226, Y 17.4415, Z -1.3333, A 0.000, B 0.000, C 0.000 }
gfCNCPoint1[1025] = {X 549.6228, Y 38.4561, Z -1.3333, A 0.000, B 0.000, C 0.000 }
gfCNCPoint1[1026] = {X 551.8213, Y 39.4186, Z -1.3333, A 0.000, B 0.000, C 0.000 }
gfCNCPoint1[1027] = {X 552.0827, Y 38.8622, Z -1.3333, A 0.000, B 0.000, C 0.000 }
gfCNCPoint1[1028] = {X 552.3730, Y 38.3204, Z -1.3333, A 0.000, B 0.000, C 0.000 }
gfCNCPoint1[1029] = {X 552.3730, Y 11.6898, Z -1.3333, A 0.000, B 0.000, C 0.000 }
gfCNCPoint1[1030] = {X 551.6711, Y 10.2350, Z -1.3333, A 0.000, B 0.000, C 0.000 }
gfCNCPoint1[1031] = {X 551.1781, Y 8.6969, Z -1.3333, A 0.000, B 0.000, C 0.000 }
gfCNCPoint1[1032] = {X 550.9036, Y 7.1051, Z -1.3333, A 0.000, B 0.000, C 0.000 }
gfCNCPoint1[1033] = {X 524.2929, Y 7.1051, Z -1.3333, A 0.000, B 0.000, C 0.000 }
gfCNCPoint1[1034] = {X 524.3791, Y 7.2071, Z -1.3333, A 0.000, B 0.000, C 0.000 }
gfCNCPoint1[1035] = {X 524.4625, Y 7.3113, Z -1.3333, A 0.000, B 0.000, C 0.000 }
gfCNCPoint1[1036] = {X 543.7427, Y 7.3119, Z -1.3333, A 0.000, B 0.000, C 0.000 }
gfCNCPoint1[1037] = {X 544.7117, Y 7.3840, Z -1.3333, A 0.000, B 0.000, C 0.000 }
gfCNCPoint1[1038] = {X 545.6473, Y 7.6465, Z -1.3333, A 0.000, B 0.000, C 0.000 }
gfCNCPoint1[1039] = {X 546.5125, Y 8.0891, Z -1.3333, A 0.000, B 0.000, C 0.000 }
gfCNCPoint1[1040] = {X 547.2729, Y 8.6940, Z -1.3333, A 0.000, B 0.000, C 0.000 }
gfCNCPoint1[1041] = {X 547.8985, Y 9.4376, Z -1.3333, A 0.000, B 0.000, C 0.000 }
gfCNCPoint1[1042] = {X 548.3646, Y 10.2903, Z -1.3333, A 0.000, B 0.000, C 0.000 }
gfCNCPoint1[1043] = {X 548.6527, Y 11.2183, Z -1.3333, A 0.000, B 0.000, C 0.000 }
gfCNCPoint1[1044] = {X 548.7514, Y 12.1850, Z -1.3333, A 0.000, B 0.000, C 0.000 }
gfCNCPoint1[1045] = {X 548.7512, Y 13.0283, Z -1.3333, A 0.000, B 0.000, C 0.000 }
gfCNCPoint1[1046] = {X 548.6549, Y 13.9436, Z -1.3333, A 0.000, B 0.000, C 0.000 }
gfCNCPoint1[1047] = {X 548.3886, Y 14.8246, Z -1.3333, A 0.000, B 0.000, C 0.000 }
gfCNCPoint1[1048] = {X 547.9615, Y 15.6399, Z -1.3333, A 0.000, B 0.000, C 0.000 }
gfCNCPoint1[1049] = {X 547.6183, Y 16.1046, Z -1.3333, A 0.000, B 0.000, C 0.000 }
gfCNCPoint1[1050] = {X 547.2226, Y 16.5254, Z -1.3333, A 0.000, B 0.000, C 0.000 }
gfCNCPoint1[1051] = {X 547.2228, Y 40.6616, Z -1.3333, A 0.000, B 0.000, C 0.000 }
gfCNCPoint1[1052] = {X 547.8646, Y 41.4037, Z -1.3333, A 0.000, B 0.000, C 0.000 }
gfCNCPoint1[1053] = {X 548.3450, Y 42.2591, Z -1.3333, A 0.000, B 0.000, C 0.000 }
gfCNCPoint1[1054] = {X 548.6446, Y 43.1934, Z -1.3333, A 0.000, B 0.000, C 0.000 }
gfCNCPoint1[1055] = {X 548.7513, Y 44.1687, Z -1.3333, A 0.000, B 0.000, C 0.000 }
gfCNCPoint1[1056] = {X 548.7514, Y 45.0018, Z -1.3333, A 0.000, B 0.000, C 0.000 }
gfCNCPoint1[1057] = {X 548.6694, Y 45.8828, Z -1.3333, A 0.000, B 0.000, C 0.000 }
gfCNCPoint1[1058] = {X 548.4298, Y 46.7346, Z -1.3333, A 0.000, B 0.000, C 0.000 }
gfCNCPoint1[1059] = {X 548.0405, Y 47.5291, Z -1.3333, A 0.000, B 0.000, C 0.000 }
gfCNCPoint1[1060] = {X 547.5142, Y 48.2404, Z -1.3333, A 0.000, B 0.000, C 0.000 }
gfCNCPoint1[1061] = {X 546.7287, Y 48.9499, Z -1.3333, A 0.000, B 0.000, C 0.000 }
gfCNCPoint1[1062] = {X 545.8087, Y 49.4735, Z -1.3333, A 0.000, B 0.000, C 0.000 }
gfCNCPoint1[1063] = {X 544.7975, Y 49.7867, Z -1.3333, A 0.000, B 0.000, C 0.000 }
gfCNCPoint1[1064] = {X 543.7426, Y 49.8746, Z -1.3333, A 0.000, B 0.000, C 0.000 }
gfCNCPoint1[1065] = {X 524.3230, Y 49.8752, Z -1.3333, A 0.000, B 0.000, C 0.000 }
gfCNCPoint1[1066] = {X 523.7103, Y 50.5141, Z -1.3333, A 0.000, B 0.000, C 0.000 }
gfCNCPoint1[1067] = {X 522.9952, Y 51.0360, Z -1.3333, A 0.000, B 0.000, C 0.000 }
gfCNCPoint1[1068] = {X 522.1998, Y 51.4247, Z -1.3333, A 0.000, B 0.000, C 0.000 }
gfCNCPoint1[1069] = {X 521.3487, Y 51.6683, Z -1.3333, A 0.000, B 0.000, C 0.000 }
gfCNCPoint1[1070] = {X 520.4681, Y 51.7591, Z -1.3333, A 0.000, B 0.000, C 0.000 }
gfCNCPoint1[1071] = {X 519.7998, Y 51.7591, Z -1.3333, A 0.000, B 0.000, C 0.000 }
gfCNCPoint1[1072] = {X 518.8477, Y 51.6654, Z -1.3333, A 0.000, B 0.000, C 0.000 }
gfCNCPoint1[1073] = {X 517.9323, Y 51.3877, Z -1.3333, A 0.000, B 0.000, C 0.000 }
gfCNCPoint1[1074] = {X 517.0886, Y 50.9367, Z -1.3333, A 0.000, B 0.000, C 0.000 }
gfCNCPoint1[1075] = {X 516.3491, Y 50.3298, Z -1.3333, A 0.000, B 0.000, C 0.000 }
gfCNCPoint1[1076] = {X 515.7422, Y 49.5903, Z -1.3333, A 0.000, B 0.000, C 0.000 }
gfCNCPoint1[1077] = {X 515.2912, Y 48.7466, Z -1.3333, A 0.000, B 0.000, C 0.000 }
gfCNCPoint1[1078] = {X 515.0135, Y 47.8312, Z -1.3333, A 0.000, B 0.000, C 0.000 }
gfCNCPoint1[1079] = {X 514.9198, Y 46.8791, Z -1.3333, A 0.000, B 0.000, C 0.000 }
gfCNCPoint1[1080] = {X 514.9198, Y 39.9011, Z -1.3333, A 0.000, B 0.000, C 0.000 }
gfCNCPoint1[1081] = {X 515.0197, Y 38.9186, Z -1.3333, A 0.000, B 0.000, C 0.000 }
gfCNCPoint1[1082] = {X 515.3154, Y 37.9764, Z -1.3333, A 0.000, B 0.000, C 0.000 }
gfCNCPoint1[1083] = {X 515.7947, Y 37.1129, Z -1.3333, A 0.000, B 0.000, C 0.000 }
gfCNCPoint1[1084] = {X 516.4381, Y 36.3637, Z -1.3333, A 0.000, B 0.000, C 0.000 }
gfCNCPoint1[1085] = {X 517.2191, Y 35.7593, Z -1.3333, A 0.000, B 0.000, C 0.000 }
gfCNCPoint1[1086] = {X 518.1058, Y 35.3245, Z -1.3333, A 0.000, B 0.000, C 0.000 }
gfCNCPoint1[1087] = {X 519.0619, Y 35.0772, Z -1.3333, A 0.000, B 0.000, C 0.000 }
gfCNCPoint1[1088] = {X 519.4084, Y 35.0368, Z -1.3333, A 0.000, B 0.000, C 0.000 }
gfCNCPoint1[1089] = {X 519.7568, Y 35.0213, Z -1.3333, A 0.000, B 0.000, C 0.000 }
gfCNCPoint1[1090] = {X 520.5345, Y 35.0216, Z -1.3333, A 0.000, B 0.000, C 0.000 }
gfCNCPoint1[1091] = {X 521.4088, Y 35.1126, Z -1.3333, A 0.000, B 0.000, C 0.000 }
gfCNCPoint1[1092] = {X 522.2525, Y 35.3590, Z -1.3333, A 0.000, B 0.000, C 0.000 }
gfCNCPoint1[1093] = {X 523.0383, Y 35.7527, Z -1.3333, A 0.000, B 0.000, C 0.000 }
gfCNCPoint1[1094] = {X 523.7407, Y 36.2811, Z -1.3333, A 0.000, B 0.000, C 0.000 }
gfCNCPoint1[1095] = {X 524.3370, Y 36.9268, Z -1.3333, A 0.000, B 0.000, C 0.000 }
gfCNCPoint1[1096] = {X 534.0719, Y 36.9274, Z -1.3333, A 0.000, B 0.000, C 0.000 }
gfCNCPoint1[1097] = {X 534.0719, Y 34.5244, Z -1.3333, A 0.000, B 0.000, C 0.000 }
gfCNCPoint1[1098] = {X 530.3971, Y 34.5240, Z -1.3333, A 0.000, B 0.000, C 0.000 }
gfCNCPoint1[1099] = {X 529.7972, Y 35.1730, Z -1.3333, A 0.000, B 0.000, C 0.000 }
gfCNCPoint1[1100] = {X 529.0900, Y 35.7031, Z -1.3333, A 0.000, B 0.000, C 0.000 }
gfCNCPoint1[1101] = {X 528.2989, Y 36.0970, Z -1.3333, A 0.000, B 0.000, C 0.000 }
gfCNCPoint1[1102] = {X 527.4497, Y 36.3417, Z -1.3333, A 0.000, B 0.000, C 0.000 }
gfCNCPoint1[1103] = {X 526.5703, Y 36.4293, Z -1.3333, A 0.000, B 0.000, C 0.000 }
gfCNCPoint1[1104] = {X 525.8868, Y 36.4294, Z -1.3333, A 0.000, B 0.000, C 0.000 }
gfCNCPoint1[1105] = {X 524.9094, Y 36.3306, Z -1.3333, A 0.000, B 0.000, C 0.000 }
gfCNCPoint1[1106] = {X 523.9717, Y 36.0380, Z -1.3333, A 0.000, B 0.000, C 0.000 }
gfCNCPoint1[1107] = {X 523.1116, Y 35.5636, Z -1.3333, A 0.000, B 0.000, C 0.000 }
gfCNCPoint1[1108] = {X 522.3639, Y 34.9265, Z -1.3333, A 0.000, B 0.000, C 0.000 }
gfCNCPoint1[1109] = {X 521.7590, Y 34.1525, Z -1.3333, A 0.000, B 0.000, C 0.000 }
gfCNCPoint1[1110] = {X 521.3213, Y 33.2731, Z -1.3333, A 0.000, B 0.000, C 0.000 }
gfCNCPoint1[1111] = {X 521.0686, Y 32.3239, Z -1.3333, A 0.000, B 0.000, C 0.000 }
gfCNCPoint1[1112] = {X 521.0222, Y 31.9379, Z -1.3333, A 0.000, B 0.000, C 0.000 }
gfCNCPoint1[1113] = {X 521.0068, Y 31.5495, Z -1.3333, A 0.000, B 0.000, C 0.000 }
gfCNCPoint1[1114] = {X 521.0076, Y 24.4815, Z -1.3333, A 0.000, B 0.000, C 0.000 }
gfCNCPoint1[1115] = {X 521.0984, Y 23.6300, Z -1.3333, A 0.000, B 0.000, C 0.000 }
gfCNCPoint1[1116] = {X 521.3368, Y 22.8074, Z -1.3333, A 0.000, B 0.000, C 0.000 }
gfCNCPoint1[1117] = {X 521.7152, Y 22.0391, Z -1.3333, A 0.000, B 0.000, C 0.000 }
gfCNCPoint1[1118] = {X 521.1864, Y 22.1316, Z -1.3333, A 0.000, B 0.000, C 0.000 }
gfCNCPoint1[1119] = {X 520.6505, Y 22.1656, Z -1.3333, A 0.000, B 0.000, C 0.000 }
gfCNCPoint1[1120] = {X 519.9691, Y 22.1657, Z -1.3333, A 0.000, B 0.000, C 0.000 }
gfCNCPoint1[1121] = {X 519.5109, Y 22.1442, Z -1.3333, A 0.000, B 0.000, C 0.000 }
gfCNCPoint1[1122] = {X 519.0567, Y 22.0797, Z -1.3333, A 0.000, B 0.000, C 0.000 }
gfCNCPoint1[1123] = {X 518.1336, Y 21.8074, Z -1.3333, A 0.000, B 0.000, C 0.000 }
gfCNCPoint1[1124] = {X 517.2820, Y 21.3592, Z -1.3333, A 0.000, B 0.000, C 0.000 }
gfCNCPoint1[1125] = {X 516.5348, Y 20.7527, Z -1.3333, A 0.000, B 0.000, C 0.000 }
gfCNCPoint1[1126] = {X 515.9212, Y 20.0113, Z -1.3333, A 0.000, B 0.000, C 0.000 }
gfCNCPoint1[1127] = {X 515.4650, Y 19.1639, Z -1.3333, A 0.000, B 0.000, C 0.000 }
gfCNCPoint1[1128] = {X 515.1840, Y 18.2434, Z -1.3333, A 0.000, B 0.000, C 0.000 }
gfCNCPoint1[1129] = {X 515.0891, Y 17.2857, Z -1.3333, A 0.000, B 0.000, C 0.000 }
gfCNCPoint1[1130] = {X 515.0891, Y 10.3077, Z -1.3333, A 0.000, B 0.000, C 0.000 }
gfCNCPoint1[1131] = {X 515.0965, Y 10.0383, Z -1.3333, A 0.000, B 0.000, C 0.000 }
gfCNCPoint1[1132] = {X 515.1189, Y 9.7697, Z -1.3333, A 0.000, B 0.000, C 0.000 }
gfCNCPoint1[1133] = {X 515.3251, Y 8.8085, Z -1.3333, A 0.000, B 0.000, C 0.000 }
gfCNCPoint1[1134] = {X 515.7198, Y 7.9081, Z -1.3333, A 0.000, B 0.000, C 0.000 }
gfCNCPoint1[1135] = {X 516.2870, Y 7.1051, Z -1.3333, A 0.000, B 0.000, C 0.000 }
gfCNCPoint1[1136] = {X 516.6492, Y 7.4201, Z -1.3333, A 0.000, B 0.000, C 0.000 }
gfCNCPoint1[1137] = {X 517.3372, Y 6.7816, Z -1.3333, A 0.000, B 0.000, C 0.000 }
gfCNCPoint1[1138] = {X 518.1451, Y 6.3036, Z -1.3333, A 0.000, B 0.000, C 0.000 }
gfCNCPoint1[1139] = {X 519.0359, Y 6.0078, Z -1.3333, A 0.000, B 0.000, C 0.000 }
gfCNCPoint1[1140] = {X 519.9693, Y 5.9077, Z -1.3333, A 0.000, B 0.000, C 0.000 }
gfCNCPoint1[1141] = {X 520.6509, Y 5.9079, Z -1.3333, A 0.000, B 0.000, C 0.000 }
gfCNCPoint1[1142] = {X 521.4836, Y 5.9951, Z -1.3333, A 0.000, B 0.000, C 0.000 }
gfCNCPoint1[1143] = {X 522.2847, Y 6.2385, Z -1.3333, A 0.000, B 0.000, C 0.000 }
gfCNCPoint1[1144] = {X 523.0251, Y 6.6293, Z -1.3333, A 0.000, B 0.000, C 0.000 }
gfCNCPoint1[1145] = {X 523.6782, Y 7.1532, Z -1.3333, A 0.000, B 0.000, C 0.000 }
gfCNCPoint1[1146] = {X 524.2202, Y 7.7913, Z -1.3333, A 0.000, B 0.000, C 0.000 }
gfCNCPoint1[1147] = {X 543.7489, Y 7.7919, Z -1.3333, A 0.000, B 0.000, C 0.000 }
gfCNCPoint1[1148] = {X 544.7469, Y 7.8792, Z -1.3333, A 0.000, B 0.000, C 0.000 }
gfCNCPoint1[1149] = {X 545.6993, Y 8.1898, Z -1.3333, A 0.000, B 0.000, C 0.000 }
gfCNCPoint1[1150] = {X 546.5569, Y 8.7075, Z -1.3333, A 0.000, B 0.000, C 0.000 }
gfCNCPoint1[1151] = {X 547.2754, Y 9.4056, Z -1.3333, A 0.000, B 0.000, C 0.000 }
gfCNCPoint1[1152] = {X 547.8176, Y 10.2479, Z -1.3333, A 0.000, B 0.000, C 0.000 }
gfCNCPoint1[1153] = {X 548.1554, Y 11.1910, Z -1.3333, A 0.000, B 0.000, C 0.000 }
gfCNCPoint1[1154] = {X 548.2714, Y 12.1860, Z -1.3333, A 0.000, B 0.000, C 0.000 }
gfCNCPoint1[1155] = {X 548.2712, Y 13.0233, Z -1.3333, A 0.000, B 0.000, C 0.000 }
gfCNCPoint1[1156] = {X 548.1628, Y 13.9498, Z -1.3333, A 0.000, B 0.000, C 0.000 }
gfCNCPoint1[1157] = {X 547.8615, Y 14.8325, Z -1.3333, A 0.000, B 0.000, C 0.000 }
gfCNCPoint1[1158] = {X 547.3809, Y 15.6320, Z -1.3333, A 0.000, B 0.000, C 0.000 }
gfCNCPoint1[1159] = {X 546.7426, Y 16.3121, Z -1.3333, A 0.000, B 0.000, C 0.000 }
gfCNCPoint1[1160] = {X 546.7428, Y 40.8749, Z -1.3333, A 0.000, B 0.000, C 0.000 }
gfCNCPoint1[1161] = {X 547.3879, Y 41.5641, Z -1.3333, A 0.000, B 0.000, C 0.000 }
gfCNCPoint1[1162] = {X 547.8711, Y 42.3750, Z -1.3333, A 0.000, B 0.000, C 0.000 }
gfCNCPoint1[1163] = {X 548.1702, Y 43.2704, Z -1.3333, A 0.000, B 0.000, C 0.000 }
gfCNCPoint1[1164] = {X 548.2714, Y 44.2089, Z -1.3333, A 0.000, B 0.000, C 0.000 }
gfCNCPoint1[1165] = {X 548.2714, Y 45.0008, Z -1.3333, A 0.000, B 0.000, C 0.000 }
gfCNCPoint1[1166] = {X 548.1554, Y 45.9958, Z -1.3333, A 0.000, B 0.000, C 0.000 }
gfCNCPoint1[1167] = {X 547.8175, Y 46.9388, Z -1.3333, A 0.000, B 0.000, C 0.000 }
gfCNCPoint1[1168] = {X 547.2754, Y 47.7812, Z -1.3333, A 0.000, B 0.000, C 0.000 }
gfCNCPoint1[1169] = {X 546.5569, Y 48.4792, Z -1.3333, A 0.000, B 0.000, C 0.000 }
gfCNCPoint1[1170] = {X 545.6992, Y 48.9969, Z -1.3333, A 0.000, B 0.000, C 0.000 }
gfCNCPoint1[1171] = {X 544.7468, Y 49.3073, Z -1.3333, A 0.000, B 0.000, C 0.000 }
gfCNCPoint1[1172] = {X 543.7489, Y 49.3946, Z -1.3333, A 0.000, B 0.000, C 0.000 }
gfCNCPoint1[1173] = {X 524.0856, Y 49.3952, Z -1.3333, A 0.000, B 0.000, C 0.000 }
gfCNCPoint1[1174] = {X 523.5290, Y 50.0303, Z -1.3333, A 0.000, B 0.000, C 0.000 }
gfCNCPoint1[1175] = {X 522.8647, Y 50.5518, Z -1.3333, A 0.000, B 0.000, C 0.000 }
gfCNCPoint1[1176] = {X 522.1157, Y 50.9419, Z -1.3333, A 0.000, B 0.000, C 0.000 }
gfCNCPoint1[1177] = {X 521.3076, Y 51.1871, Z -1.3333, A 0.000, B 0.000, C 0.000 }
gfCNCPoint1[1178] = {X 520.4681, Y 51.2791, Z -1.3333, A 0.000, B 0.000, C 0.000 }
gfCNCPoint1[1179] = {X 519.7998, Y 51.2791, Z -1.3333, A 0.000, B 0.000, C 0.000 }
gfCNCPoint1[1180] = {X 518.8207, Y 51.1688, Z -1.3333, A 0.000, B 0.000, C 0.000 }
gfCNCPoint1[1181] = {X 517.8907, Y 50.8434, Z -1.3333, A 0.000, B 0.000, C 0.000 }
gfCNCPoint1[1182] = {X 517.0564, Y 50.3192, Z -1.3333, A 0.000, B 0.000, C 0.000 }
gfCNCPoint1[1183] = {X 516.3597, Y 49.6225, Z -1.3333, A 0.000, B 0.000, C 0.000 }
gfCNCPoint1[1184] = {X 515.8355, Y 48.7882, Z -1.3333, A 0.000, B 0.000, C 0.000 }
gfCNCPoint1[1185] = {X 515.5101, Y 47.8582, Z -1.3333, A 0.000, B 0.000, C 0.000 }
gfCNCPoint1[1186] = {X 515.3998, Y 46.8791, Z -1.3333, A 0.000, B 0.000, C 0.000 }
gfCNCPoint1[1187] = {X 515.3998, Y 39.9011, Z -1.3333, A 0.000, B 0.000, C 0.000 }
gfCNCPoint1[1188] = {X 515.5101, Y 38.9220, Z -1.3333, A 0.000, B 0.000, C 0.000 }
gfCNCPoint1[1189] = {X 515.8355, Y 37.9920, Z -1.3333, A 0.000, B 0.000, C 0.000 }
gfCNCPoint1[1190] = {X 516.3597, Y 37.1577, Z -1.3333, A 0.000, B 0.000, C 0.000 }
gfCNCPoint1[1191] = {X 517.0565, Y 36.4610, Z -1.3333, A 0.000, B 0.000, C 0.000 }
gfCNCPoint1[1192] = {X 517.8907, Y 35.9368, Z -1.3333, A 0.000, B 0.000, C 0.000 }
gfCNCPoint1[1193] = {X 518.8208, Y 35.6114, Z -1.3333, A 0.000, B 0.000, C 0.000 }
gfCNCPoint1[1194] = {X 519.7999, Y 35.5011, Z -1.3333, A 0.000, B 0.000, C 0.000 }
gfCNCPoint1[1195] = {X 520.5280, Y 35.5015, Z -1.3333, A 0.000, B 0.000, C 0.000 }
gfCNCPoint1[1196] = {X 521.3617, Y 35.5928, Z -1.3333, A 0.000, B 0.000, C 0.000 }
gfCNCPoint1[1197] = {X 522.1629, Y 35.8406, Z -1.3333, A 0.000, B 0.000, C 0.000 }
gfCNCPoint1[1198] = {X 522.9025, Y 36.2359, Z -1.3333, A 0.000, B 0.000, C 0.000 }
gfCNCPoint1[1199] = {X 523.5538, Y 36.7644, Z -1.3333, A 0.000, B 0.000, C 0.000 }
gfCNCPoint1[1200] = {X 524.0929, Y 37.4068, Z -1.3333, A 0.000, B 0.000, C 0.000 }
gfCNCPoint1[1201] = {X 534.5519, Y 37.4074, Z -1.3333, A 0.000, B 0.000, C 0.000 }
gfCNCPoint1[1202] = {X 534.5519, Y 34.0445, Z -1.3333, A 0.000, B 0.000, C 0.000 }
gfCNCPoint1[1203] = {X 530.1530, Y 34.0440, Z -1.3333, A 0.000, B 0.000, C 0.000 }
gfCNCPoint1[1204] = {X 529.6053, Y 34.6947, Z -1.3333, A 0.000, B 0.000, C 0.000 }
gfCNCPoint1[1205] = {X 528.9427, Y 35.2280, Z -1.3333, A 0.000, B 0.000, C 0.000 }
gfCNCPoint1[1206] = {X 528.1898, Y 35.6237, Z -1.3333, A 0.000, B 0.000, C 0.000 }
gfCNCPoint1[1207] = {X 527.3748, Y 35.8673, Z -1.3333, A 0.000, B 0.000, C 0.000 }
gfCNCPoint1[1208] = {X 526.5282, Y 35.9495, Z -1.3333, A 0.000, B 0.000, C 0.000 }
gfCNCPoint1[1209] = {X 525.8868, Y 35.9495, Z -1.3333, A 0.000, B 0.000, C 0.000 }
gfCNCPoint1[1210] = {X 524.9077, Y 35.8391, Z -1.3333, A 0.000, B 0.000, C 0.000 }
gfCNCPoint1[1211] = {X 523.9777, Y 35.5137, Z -1.3333, A 0.000, B 0.000, C 0.000 }
gfCNCPoint1[1212] = {X 523.1434, Y 34.9895, Z -1.3333, A 0.000, B 0.000, C 0.000 }
gfCNCPoint1[1213] = {X 522.4467, Y 34.2928, Z -1.3333, A 0.000, B 0.000, C 0.000 }
gfCNCPoint1[1214] = {X 521.9225, Y 33.4585, Z -1.3333, A 0.000, B 0.000, C 0.000 }
gfCNCPoint1[1215] = {X 521.5971, Y 32.5285, Z -1.3333, A 0.000, B 0.000, C 0.000 }
gfCNCPoint1[1216] = {X 521.4868, Y 31.5495, Z -1.3333, A 0.000, B 0.000, C 0.000 }
gfCNCPoint1[1217] = {X 521.4868, Y 24.5714, Z -1.3333, A 0.000, B 0.000, C 0.000 }
gfCNCPoint1[1218] = {X 521.5971, Y 23.5923, Z -1.3333, A 0.000, B 0.000, C 0.000 }
gfCNCPoint1[1219] = {X 521.9225, Y 22.6623, Z -1.3333, A 0.000, B 0.000, C 0.000 }
gfCNCPoint1[1220] = {X 522.4467, Y 21.8281, Z -1.3333, A 0.000, B 0.000, C 0.000 }
